// TIA Portal V17 export
// export: Created 2025-03-05T08:03:03.1395906Z, ExportSetting WithDefaults, DisplayName Totally Integrated Automation Portal, DisplayVersion V17 Update 8, DisplayName TIA Portal Openness, DisplayVersion V17 Update 8, DisplayName TIA Portal Version Control Interface, DisplayVersion V17, DisplayName SINAMICS Startdrive Advanced, DisplayVersion V17 SP2, DisplayName SINAMICS Startdrive G110M, G120, G120C, G120D, G120P, G115D, DisplayVersion V17 SP2, DisplayName SINAMICS Startdrive G130, G150, S120, S150, SINAMICS MV, S210, DisplayVersion V17 SP2, DisplayName STEP 7 Professional, DisplayVersion V17 Update 8, DisplayName SINUMERIK ONE STEP 7 Toolbox, DisplayVersion V17 Update 12, DisplayName SINUMERIK 840D sl STEP 7 Toolbox, DisplayVersion V17 Update 12, DisplayName STEP 7 Safety, DisplayVersion V17 Update 6, DisplayName WinCC Advanced, DisplayVersion V17 Update 8
FUNCTION_BLOCK "FB21013_POWDER_FEEDER_HOPPER"   // FB21013, LAD
TITLE = FB21013 POWDER FEEDER HOPPER
{ S7_Optimized_Access := 'FALSE' }
VERSION : 0.1
// stored: AutoNumber false, IsIECCheckEnabled false, SetENOAutomatically false, UDAEnableTagReadback false
   VAR_INPUT
      OPTIONS_0 : Byte := 2#0000_0000;
      iGENERAL_CONDITIONS : Bool;   // GENERAL CONDITIONS
      iPF_LINE_1_NOT_READY_FAULT : Bool;   // PF NOT READY FAULT LINE 1
      iPF_PROFINET_MODE_ACTIVE_FAULT_LINE_1 : Bool;   // PF PROFINET MODE ACTIVE FAULT LINE 1
      iPF_LINE_2_NOT_READY_FAULT : Bool;   // PF NOT READY FAULT LINE 2
      iMANUAL_START_REQ_LINE_1 : Bool;
      iMANUAL_START_REQ_LINE_2 : Bool;
      iMANUAL_STOP_REQ_LINE_1 : Bool;
      iMANUAL_STOP_REQ_LINE_2 : Bool;
      iPF_INTERLOCK_INPUTS : "POWDER FEEDER INTERLOCK INPUT";
      iFEEDER_PROFINET_MODE_ACTIVE : Bool;
      iCONTROL_ON_DELAYED : Bool;   // LOCAL MACHINE ON
      iAUTO_START_REQUEST : Bool;
      iAUTO_STOP_REQUEST : Bool;
      iHMI_GAS_SETPOINT_L1 : Real;
      iHMI_GAS_SETPOINT_L2 : Real;
      iHMI_DISK_SETPOINT_L1 : Real;
      iHMI_DISK_SETPOINT_L2 : Real;
      iCNC_GAS_SETPOINT_L1 : Real;
      iCNC_GAS_SETPOINT_L2 : Real;
      iCNC_DISK_SETPOINT_L1 : Real;
      iCNC_DISK_SETPOINT_L2 : Real;
      iFEEDER_PLC_AUX_VALUES : "POWDER FEEDER PLC AUXILIAR";
   END_VAR
   VAR_OUTPUT
      oSTATION_IS_ALARMS : Bool;   // STATION IS ALARMS
      oSTATION_WARNINGS : Bool;   // STATION WARNINGS
      o_fShutdownToPF_Line1 { ExternalAccessible := 'False'; ExternalVisible := 'False'; ExternalWritable := 'False'} : Bool;
      o_fShutdownToPF_Line2 { ExternalAccessible := 'False'; ExternalVisible := 'False'; ExternalWritable := 'False'} : Bool;
      o_fFeedingAllOnCmd_Line1 { ExternalAccessible := 'False'; ExternalVisible := 'False'; ExternalWritable := 'False'} : Bool;
      o_fFeedingAllOnCmd_Line2 { ExternalAccessible := 'False'; ExternalVisible := 'False'; ExternalWritable := 'False'} : Bool;
      o_fCarriergasOnCmd_Line1 { ExternalAccessible := 'False'; ExternalVisible := 'False'; ExternalWritable := 'False'} : Bool;
      o_fCarriergasOnCmd_Line2 { ExternalAccessible := 'False'; ExternalVisible := 'False'; ExternalWritable := 'False'} : Bool;
      o_fFeedingAllOffCmd_Line1 { ExternalAccessible := 'False'; ExternalVisible := 'False'; ExternalWritable := 'False'} : Bool;
      o_fFeedingAllOffCmd_Line2 { ExternalAccessible := 'False'; ExternalVisible := 'False'; ExternalWritable := 'False'} : Bool;
      o_fCarriergasOffCmd_Line1 { ExternalAccessible := 'False'; ExternalVisible := 'False'; ExternalWritable := 'False'} : Bool;
      o_fCarriergasOffCmd_Line2 { ExternalAccessible := 'False'; ExternalVisible := 'False'; ExternalWritable := 'False'} : Bool;
      oALARM_POWDER_LINE_1_CLOGGED : Bool;   // ALARM POWDER LINE 1 CLOGGED
      oALARM_GAS_FLOW_BELOW_LOW_LIMIT_LN_1 : Bool;   // ALARM GAS FLOW BELOW LOW LIMIT LINE 1
      oALARM_DISK_SPEED_BELOW_LOW_LIMIT_LN_1 : Bool;   // ALARM DISK SPEED BELOW LOW LIMIT LINE 1
      oALARM_STIRRER_SPEED_BELOW_LOW_LIMIT_LN_1 : Bool;   // ALARM STIRRER SPEED BELOW LOW LIMIT LINE 1
      oALARM_GAS_FLOW_ABOVE_HIGH_LIMIT_LN_1 : Bool;   // ALARM GAS FLOW ABOVE HIGH LIMIT LINE 1
      oALARM_DISK_SPEED_ABOVE_HIGH_LIMIT_LN_1 : Bool;   // ALARM DISK SPEED ABOVE HIGH LIMIT LINE 1
      oALARM_STIRRER_SPEED_ABOVE_HIGH_LIMIT_LN_1 : Bool;   // ALARM STIRRER SPEED ABOVE HIGH LIMIT LINE 1
      oALARM_CARRIER_GAS_INLET_PRESSURE_TOO_LOW_LN_1 : Bool;   // ALARM CARRIER GAS INLET PRESSURE TOO LOW LINE 1
      oALARM_DISK_MOTOR_PLUGGED_IN_AND_READY_LN_1 : Bool;   // ALARM DISK MOTOR PLUGGED IN AND READY LINE 1
      oALARM_STIRRER_PLUGGED_IN_AND_READY_LN_1 : Bool;   // ALARM STIRRER PLUGGED IN AND READY LINE 1
      oALARM_COMMUNICATION_RUNNING_LN_1 : Bool;   // ALARM COMMUNICATION RUNNING LINE 1
      oALARM_FEEDER_NOT_READY_LN_1 : Bool;   // ALARM FEEDER NOT READY LINE 1
      oWARNING_GAS_FLOW_UNDER_LIMIT_LN_1 : Bool;   // WARNING GAS FLOW UNDER LIMIT LINE 1
      oWARNING_DISK_SPEED_UNDER_LIMIT_LN_1 : Bool;   // WARNING DISK SPEED UNDER LIMIT LINE 1
      oWARNING_STIRRER_SPEED_UNDER_LIMIT_LN_1 : Bool;   // WARNING STIRRER SPEED UNDER LIMIT LINE 1
      oWARNING_GAS_FLOW_OVER_LIMIT_LN_1 : Bool;   // WARNING GAS FLOW OVER LIMIT LINE 1
      oWARNING_DISK_SPEED_OVER_LIMIT_LN_1 : Bool;   // WARNING DISK SPEED OVER LIMIT LINE 1
      oWARNING_STIRRER_SPEED_OVER_LIMIT_LN_1 : Bool;   // WARNING STIRRER SPEED OVER LIMIT LINE 1
      oALARM_POWDER_LINE_2_CLOGGED : Bool;   // ALARM POWDER LINE 2 CLOGGED
      oALARM_GAS_FLOW_BELOW_LOW_LIMIT_LN_2 : Bool;   // ALARM GAS FLOW BELOW LOW LIMIT LINE 2
      oALARM_DISK_SPEED_BELOW_LOW_LIMIT_LN_2 : Bool;   // ALARM DISK SPEED BELOW LOW LIMIT LINE 2
      oALARM_STIRRER_SPEED_BELOW_LOW_LIMIT_LN_2 : Bool;   // ALARM STIRRER SPEED BELOW LOW LIMIT LINE 2
      oALARM_GAS_FLOW_ABOVE_HIGH_LIMIT_LN_2 : Bool;   // ALARM GAS FLOW ABOVE HIGH LIMIT LINE 2
      oALARM_DISK_SPEED_ABOVE_HIGH_LIMIT_LN_2 : Bool;   // ALARM DISK SPEED ABOVE HIGH LIMIT LINE 2
      oALARM_STIRRER_SPEED_ABOVE_HIGH_LIMIT_LN_2 : Bool;   // ALARM STIRRER SPEED ABOVE HIGH LIMIT LINE 2
      oALARM_CARRIER_GAS_INLET_PRESSURE_TOO_LOW_LN_2 : Bool;   // ALARM CARRIER GAS INLET PRESSURE TOO LOW LINE 2
      oALARM_DISK_MOTOR_PLUGGED_IN_AND_READY_LN_2 : Bool;   // ALARM DISK MOTOR PLUGGED IN AND READY LINE 2
      oALARM_STIRRER_PLUGGED_IN_AND_READY_LN_2 : Bool;   // ALARM STIRRER PLUGGED IN AND READY LINE 2
      oALARM_COMMUNICATION_RUNNING_LN_2 : Bool;   // ALARM COMMUNICATION RUNNING LINE 2
      oALARM_FEEDER_NOT_READY_LN_2 : Bool;   // ALARM FEEDER NOT READY LINE 2
      oWARNING_GAS_FLOW_UNDER_LIMIT_LN_2 : Bool;   // WARNING GAS FLOW UNDER LIMIT LINE 2
      oWARNING_DISK_SPEED_UNDER_LIMIT_LN_2 : Bool;   // WARNING DISK SPEED UNDER LIMIT LINE 2
      oWARNING_STIRRER_SPEED_UNDER_LIMIT_LN_2 : Bool;   // WARNING STIRRER SPEED UNDER LIMIT LINE 2
      oWARNING_GAS_FLOW_OVER_LIMIT_LN_2 : Bool;   // WARNING GAS FLOW OVER LIMIT LINE 2
      oWARNING_DISK_SPEED_OVER_LIMIT_LN_2 : Bool;   // WARNING DISK SPEED OVER LIMIT LINE 2
      oWARNING_STIRRER_SPEED_OVER_LIMIT_LN_2 : Bool;   // WARNING STIRRER SPEED OVER LIMIT LINE 2
   END_VAR
   VAR DB_SPECIFIC
      DATA : "POWDER FEEDER HOPPER";
      INPUT_SETTINGS : Struct
         UNIT_NUMBER : Int;
         FEEDER_NUMBER : Int;
      END_STRUCT;
      Fault_timer { S7_SetPoint := 'True'} : TON_TIME;
      START_DONE_LINE_1 { S7_SetPoint := 'True'} : Bool;   // START DONE LINE 1
      START_DONE_LINE_2 { S7_SetPoint := 'True'} : Bool;   // START DONE LINE 2
      STOP_SEQUENCE_ON { S7_SetPoint := 'True'} : Bool;   // HOPPER STOP SEQUENCE IS ON
      STOP_PULSE_LINE_1 : Bool;
      STOP_PULSE_LINE_2 : Bool;
      HOPPER_STATUS_LINE_1 : Byte;   // HOPPER LINE 1 STATUS
      HOPPER_STATUS_LINE_2 : Byte;   // HOPPER LINE 2 STATUS
   END_VAR
   VAR
      SWITCH_ON_SEQUENCE_LINE_1 : "FB21250_POWDER_ON_OFF_SEQUENCE";
      SWITCH_ON_SEQUENCE_LINE_2 : "FB21250_POWDER_ON_OFF_SEQUENCE";
      SWITCH_OFF_SEQUENCE_LINE_1 : "FB21250_POWDER_ON_OFF_SEQUENCE";
      SWITCH_OFF_SEQUENCE_LINE_2 : "FB21250_POWDER_ON_OFF_SEQUENCE";
   END_VAR
   VAR DB_SPECIFIC
      SWITCH_OFF_DELAY_LINE_1 { S7_SetPoint := 'True'} : TOF_TIME;
      SWITCH_OFF_DELAY_LINE_2 { S7_SetPoint := 'True'} : TOF_TIME;
   END_VAR
   VAR_TEMP
      DB_NUMBER : DInt;
      INPUTS_MASK : Byte;
      O_BYTE_0 : Struct
         LINE_1_ENABLED : Bool;
         LINE_2_ENABLED : Bool;
         SPARE : Bool;
         SPARE_1 : Bool;
         SPARE_2 : Bool;
         SPARE_3 : Bool;
         SPARE_4 : Bool;
         SPARE_5 : Bool;
      END_STRUCT;
   END_VAR
   // Fault_timer.PT := T#1s;
   // SWITCH_OFF_DELAY_LINE_1.PT := T#4s;
   // SWITCH_OFF_DELAY_LINE_2.PT := T#4s;
   VAR_TEMP   // added for the SCL form of the ladder/FBD networks
      _w1 : Bool;
      _w2 : Bool;
   END_VAR
BEGIN

NETWORK
TITLE = READ INSTANCE DB NUMBER
      L     DINO;
      +     10#800000;
      T     #DB_NUMBER;

REGION Network 2: OPTIONS
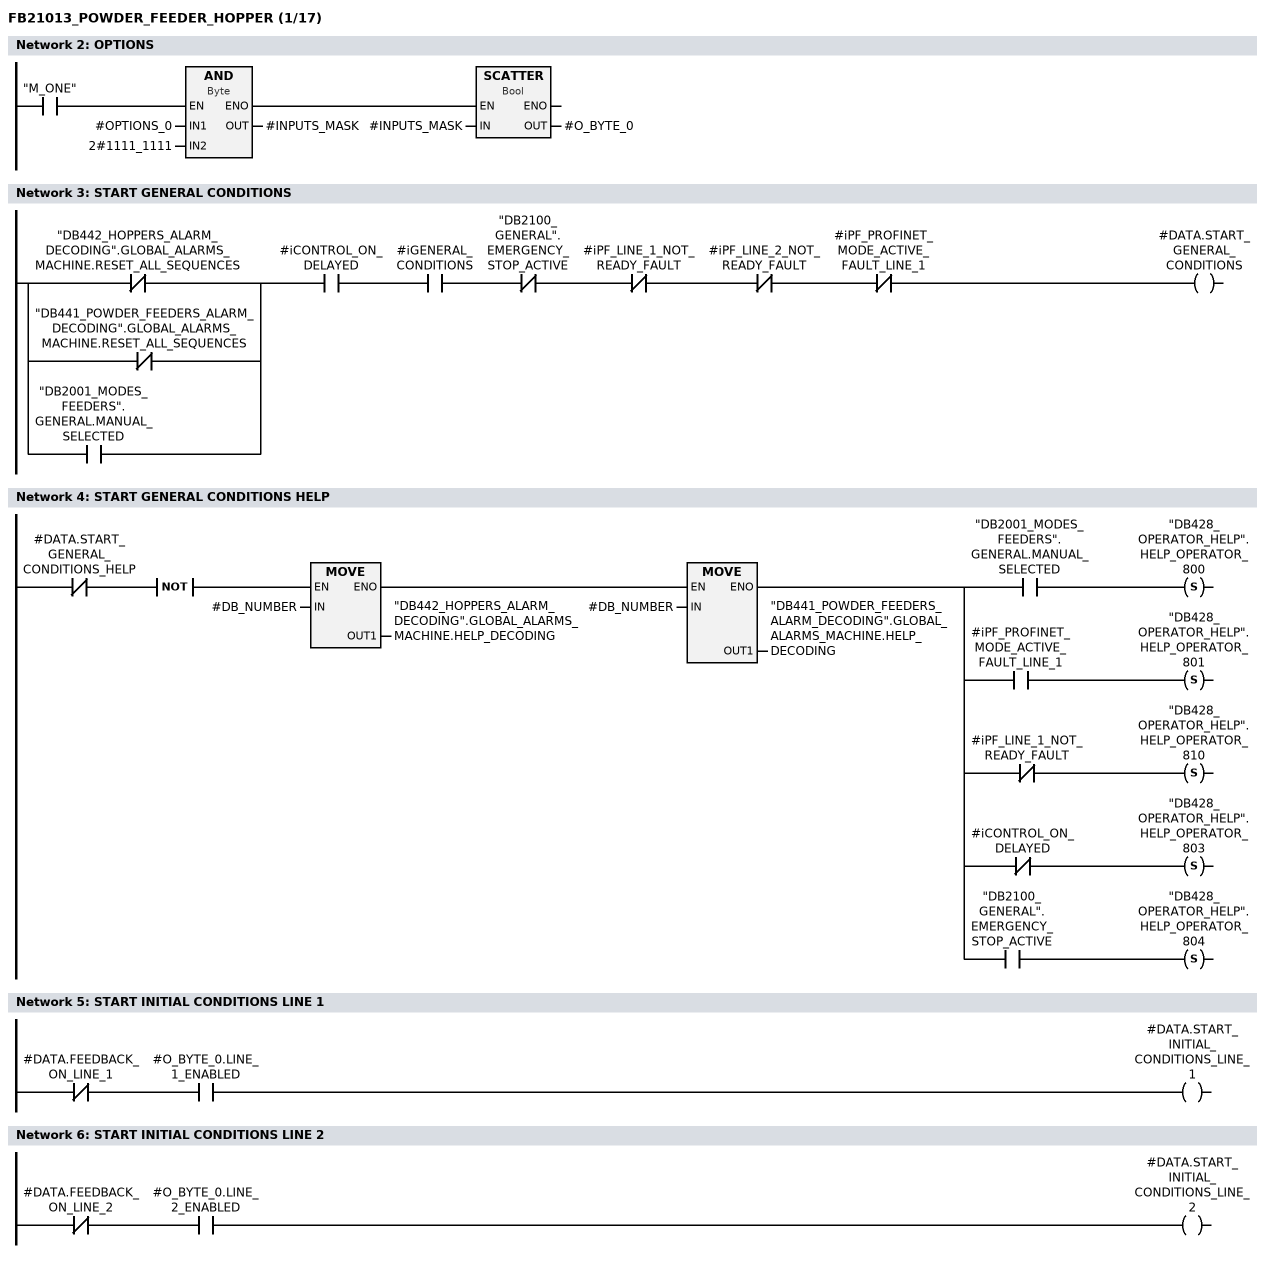
   RUNG wire#powerrail
      Contact( "M_ONE" )
      { S7_Templates := "SrcType := Byte" } And(in1 := #OPTIONS_0, in2 := 2#1111_1111, out => #INPUTS_MASK)
      { S7_Templates := "[dest_type := Bool, src_type := Byte]" } SCATTER(IN := #INPUTS_MASK, OUT => #O_BYTE_0)
   END_RUNG
   // the same network as SCL:
   IF "M_ONE" THEN
       #INPUTS_MASK := #OPTIONS_0 AND 2#1111_1111;
       SCATTER(IN := #INPUTS_MASK, OUT => #O_BYTE_0);
   END_IF;
END_REGION

REGION Network 3: START GENERAL CONDITIONS
   RUNG wire#powerrail
      I_Contact( "DB442_HOPPERS_ALARM_DECODING".GLOBAL_ALARMS_MACHINE.RESET_ALL_SEQUENCES )
      wire#w1
      Contact( #iCONTROL_ON_DELAYED )
      Contact( #iGENERAL_CONDITIONS )
      I_Contact( "DB2100_GENERAL".EMERGENCY_STOP_ACTIVE )
      I_Contact( #iPF_LINE_1_NOT_READY_FAULT )
      I_Contact( #iPF_LINE_2_NOT_READY_FAULT )
      I_Contact( #iPF_PROFINET_MODE_ACTIVE_FAULT_LINE_1 )
      Coil( #DATA.START_GENERAL_CONDITIONS )
   END_RUNG
   RUNG wire#powerrail
      I_Contact( "DB441_POWDER_FEEDERS_ALARM_DECODING".GLOBAL_ALARMS_MACHINE.RESET_ALL_SEQUENCES )
   END_RUNG wire#w1
   RUNG wire#powerrail
      Contact( "DB2001_MODES_FEEDERS".GENERAL.MANUAL_SELECTED )
   END_RUNG wire#w1
   // the same network as SCL:
   #DATA.START_GENERAL_CONDITIONS := (NOT "DB442_HOPPERS_ALARM_DECODING".GLOBAL_ALARMS_MACHINE.RESET_ALL_SEQUENCES OR NOT "DB441_POWDER_FEEDERS_ALARM_DECODING".GLOBAL_ALARMS_MACHINE.RESET_ALL_SEQUENCES OR "DB2001_MODES_FEEDERS".GENERAL.MANUAL_SELECTED) AND #iCONTROL_ON_DELAYED AND #iGENERAL_CONDITIONS AND NOT "DB2100_GENERAL".EMERGENCY_STOP_ACTIVE AND NOT #iPF_LINE_1_NOT_READY_FAULT AND NOT #iPF_LINE_2_NOT_READY_FAULT AND NOT #iPF_PROFINET_MODE_ACTIVE_FAULT_LINE_1;
END_REGION

REGION Network 4: START GENERAL CONDITIONS HELP
   RUNG wire#powerrail
      I_Contact( #DATA.START_GENERAL_CONDITIONS_HELP )
      Not()
      Move(in := #DB_NUMBER, out1 => "DB442_HOPPERS_ALARM_DECODING".GLOBAL_ALARMS_MACHINE.HELP_DECODING)
      Move(in := #DB_NUMBER, out1 => "DB441_POWDER_FEEDERS_ALARM_DECODING".GLOBAL_ALARMS_MACHINE.HELP_DECODING)
      wire#w1
      Contact( "DB2001_MODES_FEEDERS".GENERAL.MANUAL_SELECTED )
      S_Coil( "DB428_OPERATOR_HELP".HELP_OPERATOR_800 )
   END_RUNG
   RUNG wire#w1
      Contact( #iPF_PROFINET_MODE_ACTIVE_FAULT_LINE_1 )
      S_Coil( "DB428_OPERATOR_HELP".HELP_OPERATOR_801 )
   END_RUNG
   RUNG wire#w1
      I_Contact( #iPF_LINE_1_NOT_READY_FAULT )
      S_Coil( "DB428_OPERATOR_HELP".HELP_OPERATOR_810 )
   END_RUNG
   RUNG wire#w1
      I_Contact( #iCONTROL_ON_DELAYED )
      S_Coil( "DB428_OPERATOR_HELP".HELP_OPERATOR_803 )
   END_RUNG
   RUNG wire#w1
      Contact( "DB2100_GENERAL".EMERGENCY_STOP_ACTIVE )
      S_Coil( "DB428_OPERATOR_HELP".HELP_OPERATOR_804 )
   END_RUNG
   // the same network as SCL:
   #_w1 := NOT (NOT #DATA.START_GENERAL_CONDITIONS_HELP);
   IF #_w1 THEN
       "DB442_HOPPERS_ALARM_DECODING".GLOBAL_ALARMS_MACHINE.HELP_DECODING := #DB_NUMBER;
       "DB441_POWDER_FEEDERS_ALARM_DECODING".GLOBAL_ALARMS_MACHINE.HELP_DECODING := #DB_NUMBER;
   END_IF;
   IF #_w1 AND "DB2001_MODES_FEEDERS".GENERAL.MANUAL_SELECTED THEN
       "DB428_OPERATOR_HELP".HELP_OPERATOR_800 := TRUE;
   END_IF;
   IF #_w1 AND #iPF_PROFINET_MODE_ACTIVE_FAULT_LINE_1 THEN
       "DB428_OPERATOR_HELP".HELP_OPERATOR_801 := TRUE;
   END_IF;
   IF #_w1 AND NOT #iPF_LINE_1_NOT_READY_FAULT THEN "DB428_OPERATOR_HELP".HELP_OPERATOR_810 := TRUE; END_IF;
   IF #_w1 AND NOT #iCONTROL_ON_DELAYED THEN "DB428_OPERATOR_HELP".HELP_OPERATOR_803 := TRUE; END_IF;
   IF #_w1 AND "DB2100_GENERAL".EMERGENCY_STOP_ACTIVE THEN
       "DB428_OPERATOR_HELP".HELP_OPERATOR_804 := TRUE;
   END_IF;
END_REGION

REGION Network 5: START INITIAL CONDITIONS LINE 1
   RUNG wire#powerrail
      I_Contact( #DATA.FEEDBACK_ON_LINE_1 )
      Contact( #O_BYTE_0.LINE_1_ENABLED )
      Coil( #DATA.START_INITIAL_CONDITIONS_LINE_1 )
   END_RUNG
   // the same network as SCL:
   #DATA.START_INITIAL_CONDITIONS_LINE_1 := NOT #DATA.FEEDBACK_ON_LINE_1 AND #O_BYTE_0.LINE_1_ENABLED;
END_REGION

REGION Network 6: START INITIAL CONDITIONS LINE 2
   RUNG wire#powerrail
      I_Contact( #DATA.FEEDBACK_ON_LINE_2 )
      Contact( #O_BYTE_0.LINE_2_ENABLED )
      Coil( #DATA.START_INITIAL_CONDITIONS_LINE_2 )
   END_RUNG
   // the same network as SCL:
   #DATA.START_INITIAL_CONDITIONS_LINE_2 := NOT #DATA.FEEDBACK_ON_LINE_2 AND #O_BYTE_0.LINE_2_ENABLED;
END_REGION

REGION Network 7: START INITIAL CONDITIONS HELP
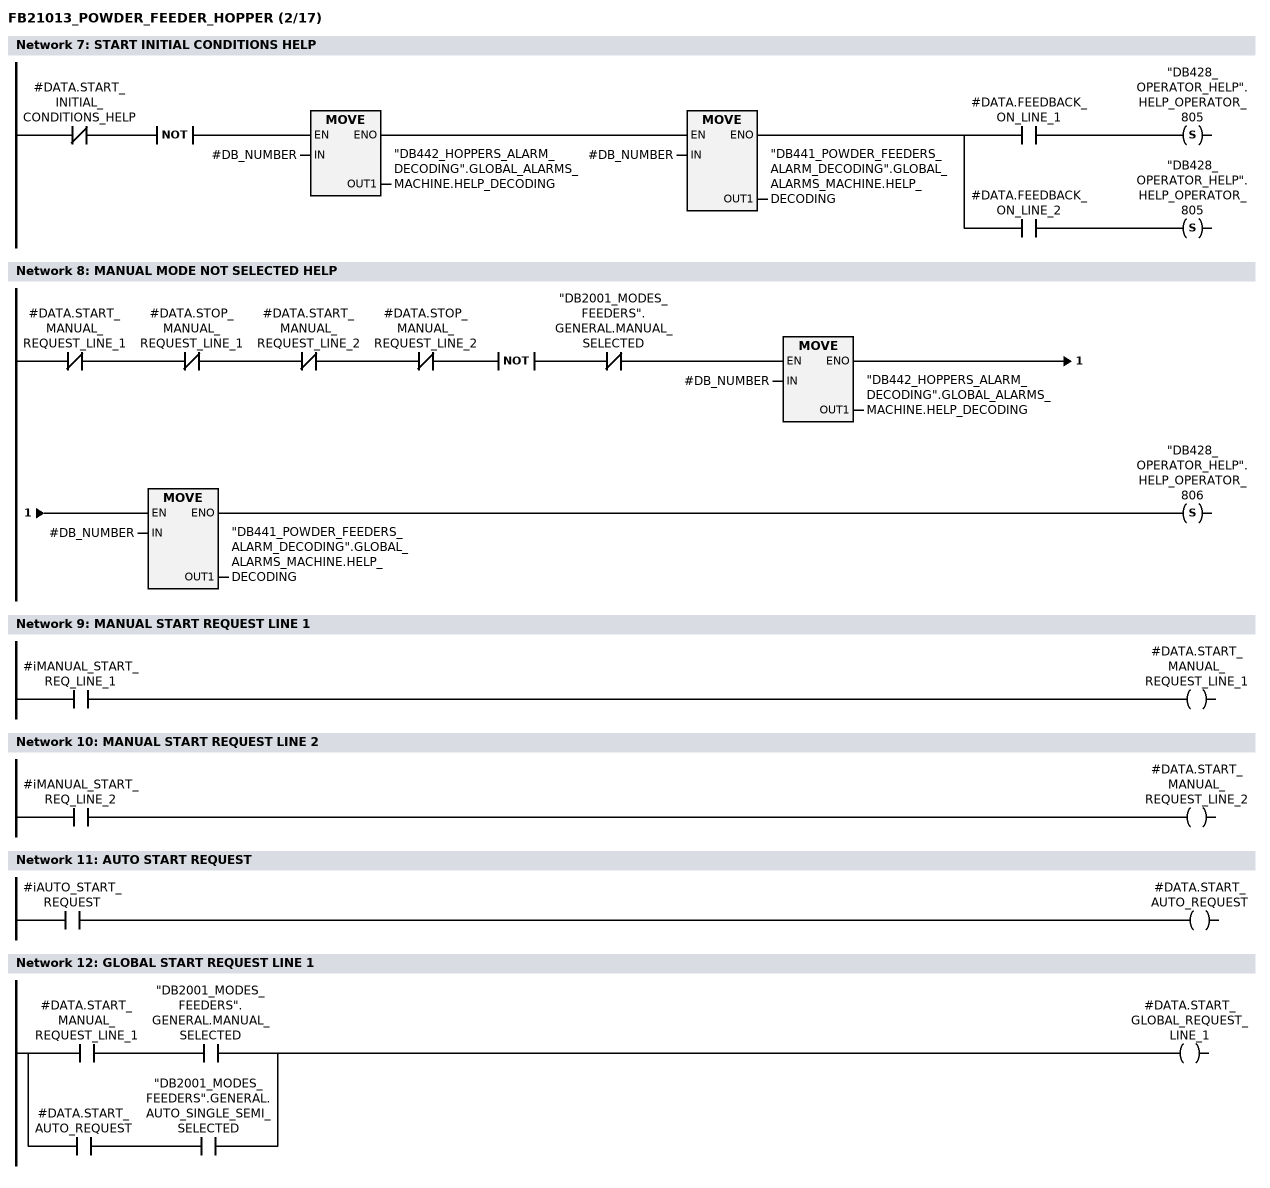
   RUNG wire#powerrail
      I_Contact( #DATA.START_INITIAL_CONDITIONS_HELP )
      Not()
      Move(in := #DB_NUMBER, out1 => "DB442_HOPPERS_ALARM_DECODING".GLOBAL_ALARMS_MACHINE.HELP_DECODING)
      Move(in := #DB_NUMBER, out1 => "DB441_POWDER_FEEDERS_ALARM_DECODING".GLOBAL_ALARMS_MACHINE.HELP_DECODING)
      wire#w1
      Contact( #DATA.FEEDBACK_ON_LINE_1 )
      S_Coil( "DB428_OPERATOR_HELP".HELP_OPERATOR_805 )
   END_RUNG
   RUNG wire#w1
      Contact( #DATA.FEEDBACK_ON_LINE_2 )
      S_Coil( "DB428_OPERATOR_HELP".HELP_OPERATOR_805 )
   END_RUNG
   // the same network as SCL:
   #_w1 := NOT (NOT #DATA.START_INITIAL_CONDITIONS_HELP);
   IF #_w1 THEN
       "DB442_HOPPERS_ALARM_DECODING".GLOBAL_ALARMS_MACHINE.HELP_DECODING := #DB_NUMBER;
       "DB441_POWDER_FEEDERS_ALARM_DECODING".GLOBAL_ALARMS_MACHINE.HELP_DECODING := #DB_NUMBER;
   END_IF;
   IF #_w1 AND #DATA.FEEDBACK_ON_LINE_1 THEN "DB428_OPERATOR_HELP".HELP_OPERATOR_805 := TRUE; END_IF;
   IF #_w1 AND #DATA.FEEDBACK_ON_LINE_2 THEN "DB428_OPERATOR_HELP".HELP_OPERATOR_805 := TRUE; END_IF;
END_REGION

REGION Network 8: MANUAL MODE NOT SELECTED HELP
   RUNG wire#powerrail
      I_Contact( #DATA.START_MANUAL_REQUEST_LINE_1 )
      I_Contact( #DATA.STOP_MANUAL_REQUEST_LINE_1 )
      I_Contact( #DATA.START_MANUAL_REQUEST_LINE_2 )
      I_Contact( #DATA.STOP_MANUAL_REQUEST_LINE_2 )
      Not()
      I_Contact( "DB2001_MODES_FEEDERS".GENERAL.MANUAL_SELECTED )
      Move(in := #DB_NUMBER, out1 => "DB442_HOPPERS_ALARM_DECODING".GLOBAL_ALARMS_MACHINE.HELP_DECODING)
      Move(in := #DB_NUMBER, out1 => "DB441_POWDER_FEEDERS_ALARM_DECODING".GLOBAL_ALARMS_MACHINE.HELP_DECODING)
      S_Coil( "DB428_OPERATOR_HELP".HELP_OPERATOR_806 )
   END_RUNG
   // the same network as SCL:
   IF NOT (NOT #DATA.START_MANUAL_REQUEST_LINE_1 AND NOT #DATA.STOP_MANUAL_REQUEST_LINE_1 AND NOT #DATA.START_MANUAL_REQUEST_LINE_2 AND NOT #DATA.STOP_MANUAL_REQUEST_LINE_2) AND NOT "DB2001_MODES_FEEDERS".GENERAL.MANUAL_SELECTED THEN
       "DB442_HOPPERS_ALARM_DECODING".GLOBAL_ALARMS_MACHINE.HELP_DECODING := #DB_NUMBER;
       "DB441_POWDER_FEEDERS_ALARM_DECODING".GLOBAL_ALARMS_MACHINE.HELP_DECODING := #DB_NUMBER;
       "DB428_OPERATOR_HELP".HELP_OPERATOR_806 := TRUE;
   END_IF;
END_REGION

REGION Network 9: MANUAL START REQUEST LINE 1
   RUNG wire#powerrail
      Contact( #iMANUAL_START_REQ_LINE_1 )
      Coil( #DATA.START_MANUAL_REQUEST_LINE_1 )
   END_RUNG
   // the same network as SCL:
   #DATA.START_MANUAL_REQUEST_LINE_1 := #iMANUAL_START_REQ_LINE_1;
END_REGION

REGION Network 10: MANUAL START REQUEST LINE 2
   RUNG wire#powerrail
      Contact( #iMANUAL_START_REQ_LINE_2 )
      Coil( #DATA.START_MANUAL_REQUEST_LINE_2 )
   END_RUNG
   // the same network as SCL:
   #DATA.START_MANUAL_REQUEST_LINE_2 := #iMANUAL_START_REQ_LINE_2;
END_REGION

REGION Network 11: AUTO START REQUEST
   RUNG wire#powerrail
      Contact( #iAUTO_START_REQUEST )
      Coil( #DATA.START_AUTO_REQUEST )
   END_RUNG
   // the same network as SCL:
   #DATA.START_AUTO_REQUEST := #iAUTO_START_REQUEST;
END_REGION

REGION Network 12: GLOBAL START REQUEST LINE 1
   RUNG wire#powerrail
      Contact( #DATA.START_MANUAL_REQUEST_LINE_1 )
      Contact( "DB2001_MODES_FEEDERS".GENERAL.MANUAL_SELECTED )
      wire#w1
      Coil( #DATA.START_GLOBAL_REQUEST_LINE_1 )
   END_RUNG
   RUNG wire#powerrail
      Contact( #DATA.START_AUTO_REQUEST )
      Contact( "DB2001_MODES_FEEDERS".GENERAL.AUTO_SINGLE_SEMI_SELECTED )
   END_RUNG wire#w1
   // the same network as SCL:
   #DATA.START_GLOBAL_REQUEST_LINE_1 := (#DATA.START_MANUAL_REQUEST_LINE_1 AND "DB2001_MODES_FEEDERS".GENERAL.MANUAL_SELECTED) OR (#DATA.START_AUTO_REQUEST AND "DB2001_MODES_FEEDERS".GENERAL.AUTO_SINGLE_SEMI_SELECTED);
END_REGION

REGION Network 13: GLOBAL START REQUEST LINE 2
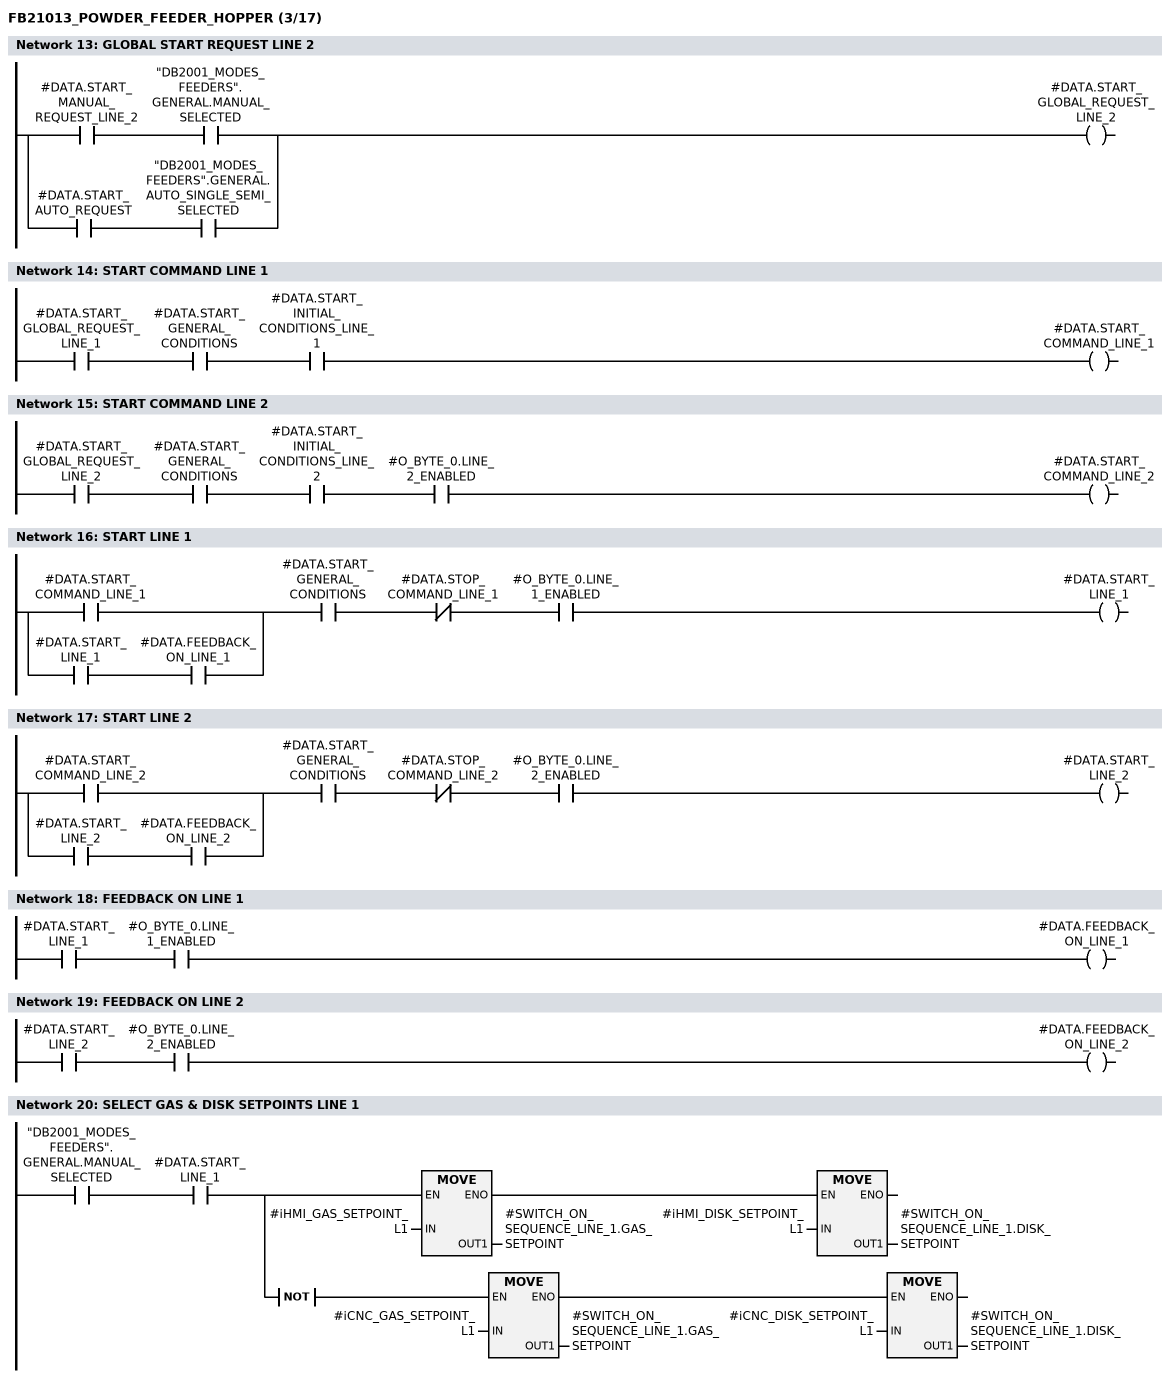
   RUNG wire#powerrail
      Contact( #DATA.START_MANUAL_REQUEST_LINE_2 )
      Contact( "DB2001_MODES_FEEDERS".GENERAL.MANUAL_SELECTED )
      wire#w1
      Coil( #DATA.START_GLOBAL_REQUEST_LINE_2 )
   END_RUNG
   RUNG wire#powerrail
      Contact( #DATA.START_AUTO_REQUEST )
      Contact( "DB2001_MODES_FEEDERS".GENERAL.AUTO_SINGLE_SEMI_SELECTED )
   END_RUNG wire#w1
   // the same network as SCL:
   #DATA.START_GLOBAL_REQUEST_LINE_2 := (#DATA.START_MANUAL_REQUEST_LINE_2 AND "DB2001_MODES_FEEDERS".GENERAL.MANUAL_SELECTED) OR (#DATA.START_AUTO_REQUEST AND "DB2001_MODES_FEEDERS".GENERAL.AUTO_SINGLE_SEMI_SELECTED);
END_REGION

REGION Network 14: START COMMAND LINE 1
   RUNG wire#powerrail
      Contact( #DATA.START_GLOBAL_REQUEST_LINE_1 )
      Contact( #DATA.START_GENERAL_CONDITIONS )
      Contact( #DATA.START_INITIAL_CONDITIONS_LINE_1 )
      Coil( #DATA.START_COMMAND_LINE_1 )
   END_RUNG
   // the same network as SCL:
   #DATA.START_COMMAND_LINE_1 := #DATA.START_GLOBAL_REQUEST_LINE_1 AND #DATA.START_GENERAL_CONDITIONS AND #DATA.START_INITIAL_CONDITIONS_LINE_1;
END_REGION

REGION Network 15: START COMMAND LINE 2
   RUNG wire#powerrail
      Contact( #DATA.START_GLOBAL_REQUEST_LINE_2 )
      Contact( #DATA.START_GENERAL_CONDITIONS )
      Contact( #DATA.START_INITIAL_CONDITIONS_LINE_2 )
      Contact( #O_BYTE_0.LINE_2_ENABLED )
      Coil( #DATA.START_COMMAND_LINE_2 )
   END_RUNG
   // the same network as SCL:
   #DATA.START_COMMAND_LINE_2 := #DATA.START_GLOBAL_REQUEST_LINE_2 AND #DATA.START_GENERAL_CONDITIONS AND #DATA.START_INITIAL_CONDITIONS_LINE_2 AND #O_BYTE_0.LINE_2_ENABLED;
END_REGION

REGION Network 16: START LINE 1
   RUNG wire#powerrail
      Contact( #DATA.START_COMMAND_LINE_1 )
      wire#w1
      Contact( #DATA.START_GENERAL_CONDITIONS )
      I_Contact( #DATA.STOP_COMMAND_LINE_1 )
      Contact( #O_BYTE_0.LINE_1_ENABLED )
      Coil( #DATA.START_LINE_1 )
   END_RUNG
   RUNG wire#powerrail
      Contact( #DATA.START_LINE_1 )
      Contact( #DATA.FEEDBACK_ON_LINE_1 )
   END_RUNG wire#w1
   // the same network as SCL:
   #DATA.START_LINE_1 := (#DATA.START_COMMAND_LINE_1 OR (#DATA.START_LINE_1 AND #DATA.FEEDBACK_ON_LINE_1)) AND #DATA.START_GENERAL_CONDITIONS AND NOT #DATA.STOP_COMMAND_LINE_1 AND #O_BYTE_0.LINE_1_ENABLED;
END_REGION

REGION Network 17: START LINE 2
   RUNG wire#powerrail
      Contact( #DATA.START_COMMAND_LINE_2 )
      wire#w1
      Contact( #DATA.START_GENERAL_CONDITIONS )
      I_Contact( #DATA.STOP_COMMAND_LINE_2 )
      Contact( #O_BYTE_0.LINE_2_ENABLED )
      Coil( #DATA.START_LINE_2 )
   END_RUNG
   RUNG wire#powerrail
      Contact( #DATA.START_LINE_2 )
      Contact( #DATA.FEEDBACK_ON_LINE_2 )
   END_RUNG wire#w1
   // the same network as SCL:
   #DATA.START_LINE_2 := (#DATA.START_COMMAND_LINE_2 OR (#DATA.START_LINE_2 AND #DATA.FEEDBACK_ON_LINE_2)) AND #DATA.START_GENERAL_CONDITIONS AND NOT #DATA.STOP_COMMAND_LINE_2 AND #O_BYTE_0.LINE_2_ENABLED;
END_REGION

REGION Network 18: FEEDBACK ON LINE 1
   RUNG wire#powerrail
      Contact( #DATA.START_LINE_1 )
      Contact( #O_BYTE_0.LINE_1_ENABLED )
      Coil( #DATA.FEEDBACK_ON_LINE_1 )
   END_RUNG
   // the same network as SCL:
   #DATA.FEEDBACK_ON_LINE_1 := #DATA.START_LINE_1 AND #O_BYTE_0.LINE_1_ENABLED;
END_REGION

REGION Network 19: FEEDBACK ON LINE 2
   RUNG wire#powerrail
      Contact( #DATA.START_LINE_2 )
      Contact( #O_BYTE_0.LINE_2_ENABLED )
      Coil( #DATA.FEEDBACK_ON_LINE_2 )
   END_RUNG
   // the same network as SCL:
   #DATA.FEEDBACK_ON_LINE_2 := #DATA.START_LINE_2 AND #O_BYTE_0.LINE_2_ENABLED;
END_REGION

REGION Network 20: SELECT GAS & DISK SETPOINTS LINE 1
   RUNG wire#powerrail
      Contact( "DB2001_MODES_FEEDERS".GENERAL.MANUAL_SELECTED )
      Contact( #DATA.START_LINE_1 )
      wire#w1
      Move(in := #iHMI_GAS_SETPOINT_L1, out1 => #SWITCH_ON_SEQUENCE_LINE_1.GAS_SETPOINT)
      Move(in := #iHMI_DISK_SETPOINT_L1, out1 => #SWITCH_ON_SEQUENCE_LINE_1.DISK_SETPOINT)
   END_RUNG
   RUNG wire#w1
      Not()
      Move(in := #iCNC_GAS_SETPOINT_L1, out1 => #SWITCH_ON_SEQUENCE_LINE_1.GAS_SETPOINT)
      Move(in := #iCNC_DISK_SETPOINT_L1, out1 => #SWITCH_ON_SEQUENCE_LINE_1.DISK_SETPOINT)
   END_RUNG
   // the same network as SCL:
   #_w1 := "DB2001_MODES_FEEDERS".GENERAL.MANUAL_SELECTED AND #DATA.START_LINE_1;
   IF #_w1 THEN
       #SWITCH_ON_SEQUENCE_LINE_1.GAS_SETPOINT := #iHMI_GAS_SETPOINT_L1;
       #SWITCH_ON_SEQUENCE_LINE_1.DISK_SETPOINT := #iHMI_DISK_SETPOINT_L1;
   END_IF;
   IF NOT #_w1 THEN
       #SWITCH_ON_SEQUENCE_LINE_1.GAS_SETPOINT := #iCNC_GAS_SETPOINT_L1;
       #SWITCH_ON_SEQUENCE_LINE_1.DISK_SETPOINT := #iCNC_DISK_SETPOINT_L1;
   END_IF;
END_REGION

REGION Network 21: SELECT GAS & DISK SETPOINTS LINE 2
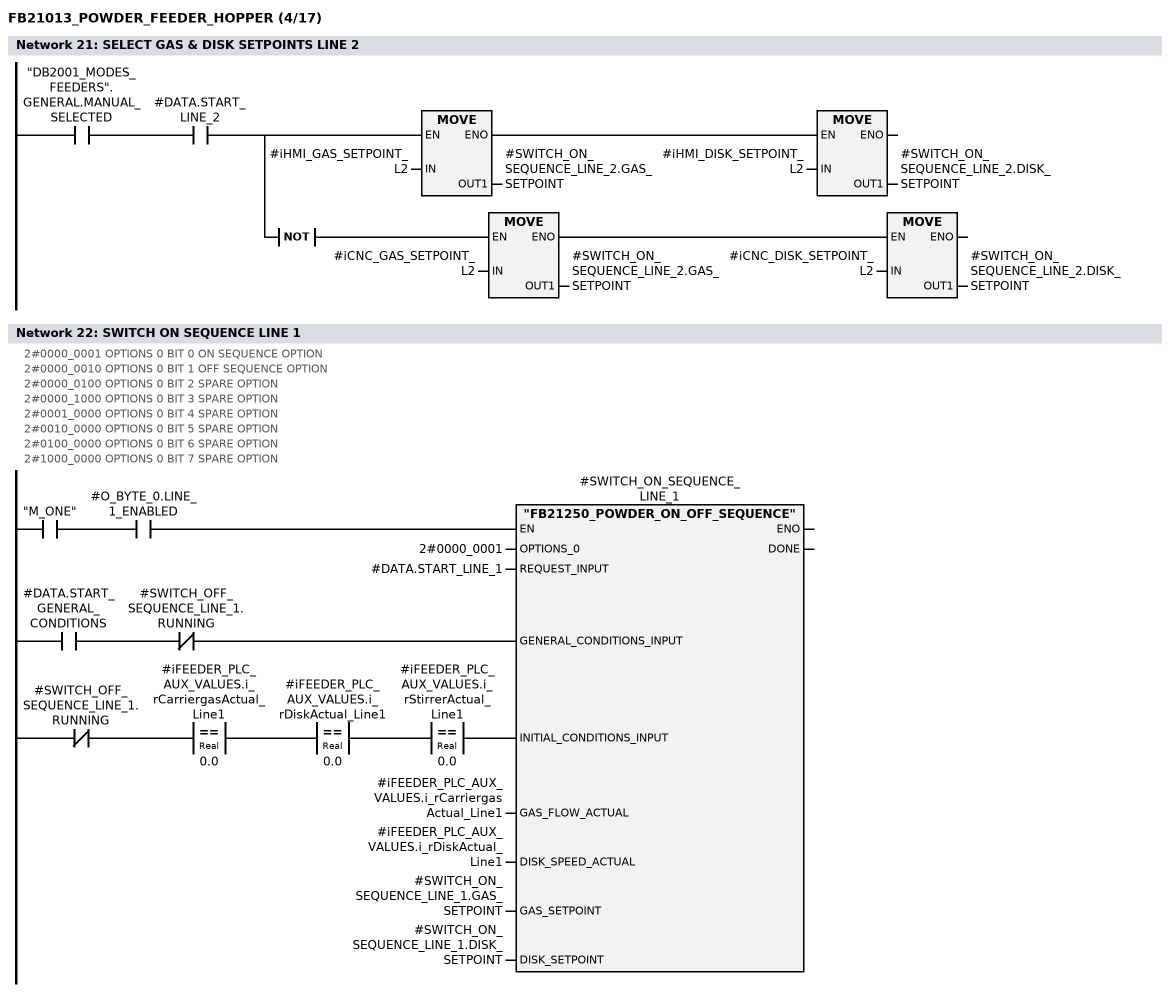
   RUNG wire#powerrail
      Contact( "DB2001_MODES_FEEDERS".GENERAL.MANUAL_SELECTED )
      Contact( #DATA.START_LINE_2 )
      wire#w1
      Move(in := #iHMI_GAS_SETPOINT_L2, out1 => #SWITCH_ON_SEQUENCE_LINE_2.GAS_SETPOINT)
      Move(in := #iHMI_DISK_SETPOINT_L2, out1 => #SWITCH_ON_SEQUENCE_LINE_2.DISK_SETPOINT)
   END_RUNG
   RUNG wire#w1
      Not()
      Move(in := #iCNC_GAS_SETPOINT_L2, out1 => #SWITCH_ON_SEQUENCE_LINE_2.GAS_SETPOINT)
      Move(in := #iCNC_DISK_SETPOINT_L2, out1 => #SWITCH_ON_SEQUENCE_LINE_2.DISK_SETPOINT)
   END_RUNG
   // the same network as SCL:
   #_w1 := "DB2001_MODES_FEEDERS".GENERAL.MANUAL_SELECTED AND #DATA.START_LINE_2;
   IF #_w1 THEN
       #SWITCH_ON_SEQUENCE_LINE_2.GAS_SETPOINT := #iHMI_GAS_SETPOINT_L2;
       #SWITCH_ON_SEQUENCE_LINE_2.DISK_SETPOINT := #iHMI_DISK_SETPOINT_L2;
   END_IF;
   IF NOT #_w1 THEN
       #SWITCH_ON_SEQUENCE_LINE_2.GAS_SETPOINT := #iCNC_GAS_SETPOINT_L2;
       #SWITCH_ON_SEQUENCE_LINE_2.DISK_SETPOINT := #iCNC_DISK_SETPOINT_L2;
   END_IF;
END_REGION

REGION Network 22: SWITCH ON SEQUENCE LINE 1
   // 2#0000_0001 OPTIONS 0 BIT 0 ON SEQUENCE OPTION
   // 2#0000_0010 OPTIONS 0 BIT 1 OFF SEQUENCE OPTION
   // 2#0000_0100 OPTIONS 0 BIT 2 SPARE OPTION
   // 2#0000_1000 OPTIONS 0 BIT 3 SPARE OPTION
   // 2#0001_0000 OPTIONS 0 BIT 4 SPARE OPTION
   // 2#0010_0000 OPTIONS 0 BIT 5 SPARE OPTION
   // 2#0100_0000 OPTIONS 0 BIT 6 SPARE OPTION
   // 2#1000_0000 OPTIONS 0 BIT 7 SPARE OPTION
   RUNG wire#powerrail
      Contact( "M_ONE" )
      Contact( #O_BYTE_0.LINE_1_ENABLED )
      #SWITCH_ON_SEQUENCE_LINE_1(GENERAL_CONDITIONS_INPUT := wire#w1, INITIAL_CONDITIONS_INPUT := wire#w2, OPTIONS_0 := 2#0000_0001, REQUEST_INPUT := #DATA.START_LINE_1, GAS_FLOW_ACTUAL := #iFEEDER_PLC_AUX_VALUES.i_rCarriergasActual_Line1, DISK_SPEED_ACTUAL := #iFEEDER_PLC_AUX_VALUES.i_rDiskActual_Line1, GAS_SETPOINT := #SWITCH_ON_SEQUENCE_LINE_1.GAS_SETPOINT, DISK_SETPOINT := #SWITCH_ON_SEQUENCE_LINE_1.DISK_SETPOINT, DONE =>)
   END_RUNG
   RUNG wire#powerrail
      Contact( #DATA.START_GENERAL_CONDITIONS )
      I_Contact( #SWITCH_OFF_SEQUENCE_LINE_1.RUNNING )
   END_RUNG wire#w1
   RUNG wire#powerrail
      I_Contact( #SWITCH_OFF_SEQUENCE_LINE_1.RUNNING )
      { S7_Templates := "SrcType := Real" } EQ_Contact(in1 := #iFEEDER_PLC_AUX_VALUES.i_rCarriergasActual_Line1, in2 := 0.0)
      { S7_Templates := "SrcType := Real" } EQ_Contact(in1 := #iFEEDER_PLC_AUX_VALUES.i_rDiskActual_Line1, in2 := 0.0)
      { S7_Templates := "SrcType := Real" } EQ_Contact(in1 := #iFEEDER_PLC_AUX_VALUES.i_rStirrerActual_Line1, in2 := 0.0)
   END_RUNG wire#w2
   // the same network as SCL:
   IF "M_ONE" AND #O_BYTE_0.LINE_1_ENABLED THEN
       #SWITCH_ON_SEQUENCE_LINE_1(OPTIONS_0 := 2#0000_0001,   // "FB21250_POWDER_ON_OFF_SEQUENCE"
                               REQUEST_INPUT := #DATA.START_LINE_1,
                               GENERAL_CONDITIONS_INPUT := #DATA.START_GENERAL_CONDITIONS AND NOT #SWITCH_OFF_SEQUENCE_LINE_1.RUNNING,
                               INITIAL_CONDITIONS_INPUT := NOT #SWITCH_OFF_SEQUENCE_LINE_1.RUNNING AND (#iFEEDER_PLC_AUX_VALUES.i_rCarriergasActual_Line1 = 0.0) AND (#iFEEDER_PLC_AUX_VALUES.i_rDiskActual_Line1 = 0.0) AND (#iFEEDER_PLC_AUX_VALUES.i_rStirrerActual_Line1 = 0.0),
                               GAS_FLOW_ACTUAL := #iFEEDER_PLC_AUX_VALUES.i_rCarriergasActual_Line1,
                               DISK_SPEED_ACTUAL := #iFEEDER_PLC_AUX_VALUES.i_rDiskActual_Line1,
                               GAS_SETPOINT := #SWITCH_ON_SEQUENCE_LINE_1.GAS_SETPOINT,
                               DISK_SETPOINT := #SWITCH_ON_SEQUENCE_LINE_1.DISK_SETPOINT);
   END_IF;
END_REGION

REGION Network 23: SWITCH ON SEQUENCE LINE 2
   // 2#0000_0001 OPTIONS 0 BIT 0 ON SEQUENCE OPTION
   // 2#0000_0010 OPTIONS 0 BIT 1 OFF SEQUENCE OPTION
   // 2#0000_0100 OPTIONS 0 BIT 2 SPARE OPTION
   // 2#0000_1000 OPTIONS 0 BIT 3 SPARE OPTION
   // 2#0001_0000 OPTIONS 0 BIT 4 SPARE OPTION
   // 2#0010_0000 OPTIONS 0 BIT 5 SPARE OPTION
   // 2#0100_0000 OPTIONS 0 BIT 6 SPARE OPTION
   // 2#1000_0000 OPTIONS 0 BIT 7 SPARE OPTION
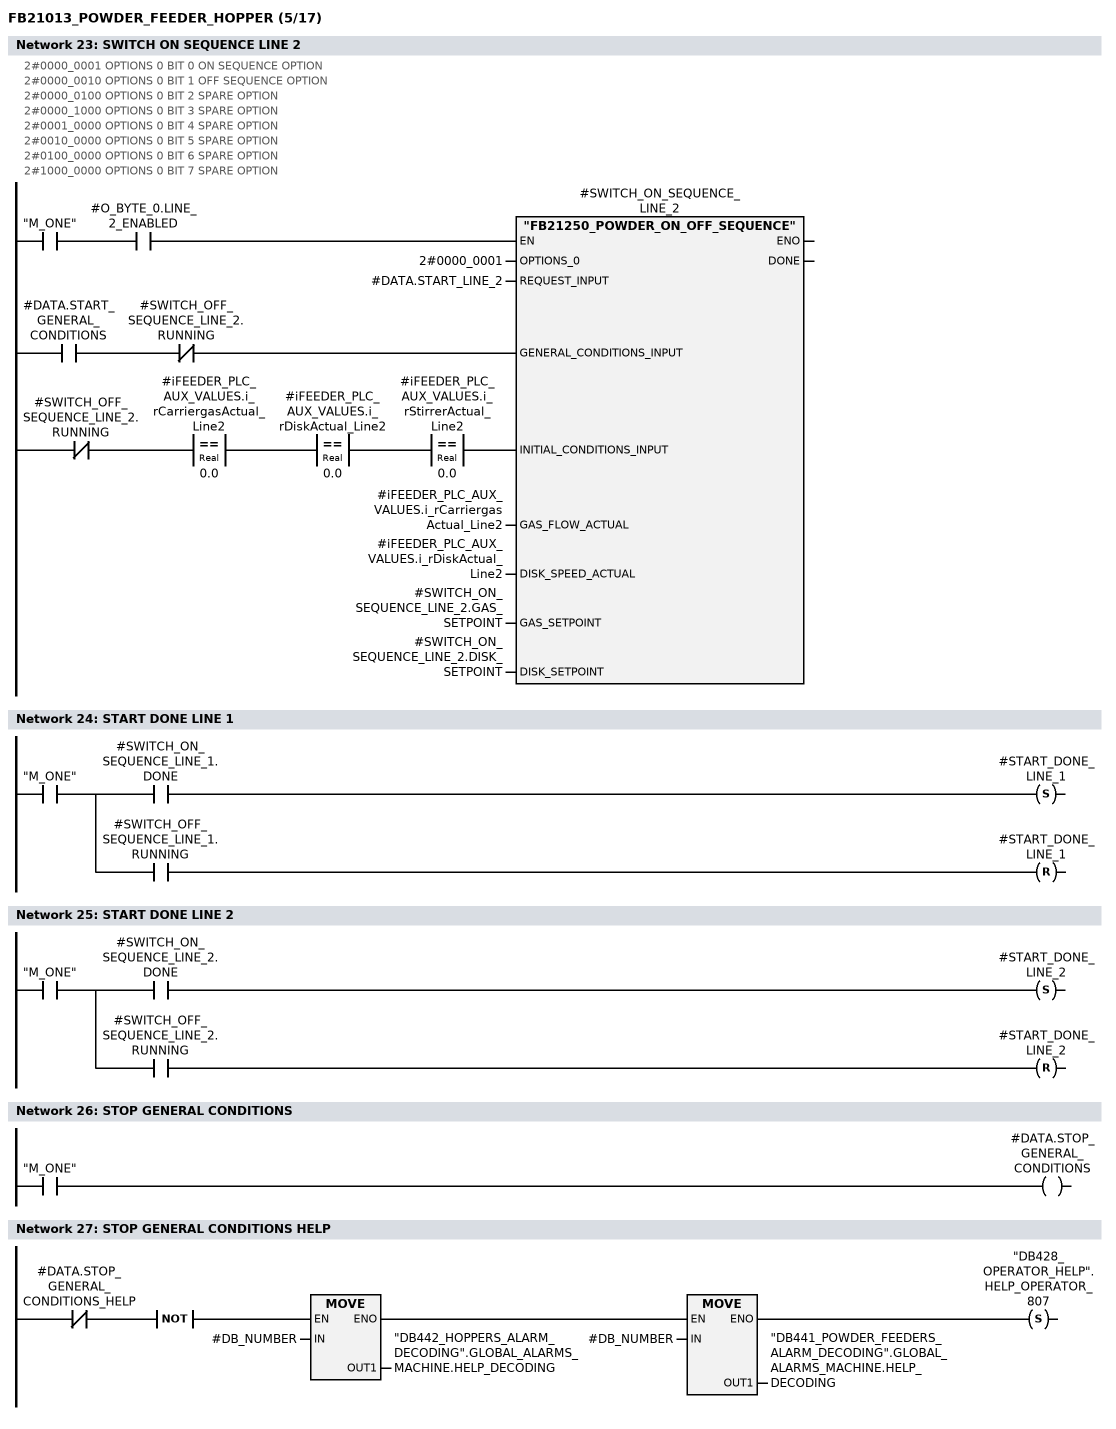
   RUNG wire#powerrail
      Contact( "M_ONE" )
      Contact( #O_BYTE_0.LINE_2_ENABLED )
      #SWITCH_ON_SEQUENCE_LINE_2(GENERAL_CONDITIONS_INPUT := wire#w1, INITIAL_CONDITIONS_INPUT := wire#w2, OPTIONS_0 := 2#0000_0001, REQUEST_INPUT := #DATA.START_LINE_2, GAS_FLOW_ACTUAL := #iFEEDER_PLC_AUX_VALUES.i_rCarriergasActual_Line2, DISK_SPEED_ACTUAL := #iFEEDER_PLC_AUX_VALUES.i_rDiskActual_Line2, GAS_SETPOINT := #SWITCH_ON_SEQUENCE_LINE_2.GAS_SETPOINT, DISK_SETPOINT := #SWITCH_ON_SEQUENCE_LINE_2.DISK_SETPOINT, DONE =>)
   END_RUNG
   RUNG wire#powerrail
      Contact( #DATA.START_GENERAL_CONDITIONS )
      I_Contact( #SWITCH_OFF_SEQUENCE_LINE_2.RUNNING )
   END_RUNG wire#w1
   RUNG wire#powerrail
      I_Contact( #SWITCH_OFF_SEQUENCE_LINE_2.RUNNING )
      { S7_Templates := "SrcType := Real" } EQ_Contact(in1 := #iFEEDER_PLC_AUX_VALUES.i_rCarriergasActual_Line2, in2 := 0.0)
      { S7_Templates := "SrcType := Real" } EQ_Contact(in1 := #iFEEDER_PLC_AUX_VALUES.i_rDiskActual_Line2, in2 := 0.0)
      { S7_Templates := "SrcType := Real" } EQ_Contact(in1 := #iFEEDER_PLC_AUX_VALUES.i_rStirrerActual_Line2, in2 := 0.0)
   END_RUNG wire#w2
   // the same network as SCL:
   IF "M_ONE" AND #O_BYTE_0.LINE_2_ENABLED THEN
       #SWITCH_ON_SEQUENCE_LINE_2(OPTIONS_0 := 2#0000_0001,   // "FB21250_POWDER_ON_OFF_SEQUENCE"
                               REQUEST_INPUT := #DATA.START_LINE_2,
                               GENERAL_CONDITIONS_INPUT := #DATA.START_GENERAL_CONDITIONS AND NOT #SWITCH_OFF_SEQUENCE_LINE_2.RUNNING,
                               INITIAL_CONDITIONS_INPUT := NOT #SWITCH_OFF_SEQUENCE_LINE_2.RUNNING AND (#iFEEDER_PLC_AUX_VALUES.i_rCarriergasActual_Line2 = 0.0) AND (#iFEEDER_PLC_AUX_VALUES.i_rDiskActual_Line2 = 0.0) AND (#iFEEDER_PLC_AUX_VALUES.i_rStirrerActual_Line2 = 0.0),
                               GAS_FLOW_ACTUAL := #iFEEDER_PLC_AUX_VALUES.i_rCarriergasActual_Line2,
                               DISK_SPEED_ACTUAL := #iFEEDER_PLC_AUX_VALUES.i_rDiskActual_Line2,
                               GAS_SETPOINT := #SWITCH_ON_SEQUENCE_LINE_2.GAS_SETPOINT,
                               DISK_SETPOINT := #SWITCH_ON_SEQUENCE_LINE_2.DISK_SETPOINT);
   END_IF;
END_REGION

REGION Network 24: START DONE LINE 1
   RUNG wire#powerrail
      Contact( "M_ONE" )
      wire#w1
      Contact( #SWITCH_ON_SEQUENCE_LINE_1.DONE )
      S_Coil( #START_DONE_LINE_1 )
   END_RUNG
   RUNG wire#w1
      Contact( #SWITCH_OFF_SEQUENCE_LINE_1.RUNNING )
      R_Coil( #START_DONE_LINE_1 )
   END_RUNG
   // the same network as SCL:
   IF "M_ONE" AND #SWITCH_ON_SEQUENCE_LINE_1.DONE THEN #START_DONE_LINE_1 := TRUE; END_IF;
   IF "M_ONE" AND #SWITCH_OFF_SEQUENCE_LINE_1.RUNNING THEN #START_DONE_LINE_1 := FALSE; END_IF;
END_REGION

REGION Network 25: START DONE LINE 2
   RUNG wire#powerrail
      Contact( "M_ONE" )
      wire#w1
      Contact( #SWITCH_ON_SEQUENCE_LINE_2.DONE )
      S_Coil( #START_DONE_LINE_2 )
   END_RUNG
   RUNG wire#w1
      Contact( #SWITCH_OFF_SEQUENCE_LINE_2.RUNNING )
      R_Coil( #START_DONE_LINE_2 )
   END_RUNG
   // the same network as SCL:
   IF "M_ONE" AND #SWITCH_ON_SEQUENCE_LINE_2.DONE THEN #START_DONE_LINE_2 := TRUE; END_IF;
   IF "M_ONE" AND #SWITCH_OFF_SEQUENCE_LINE_2.RUNNING THEN #START_DONE_LINE_2 := FALSE; END_IF;
END_REGION

REGION Network 26: STOP GENERAL CONDITIONS
   RUNG wire#powerrail
      Contact( "M_ONE" )
      Coil( #DATA.STOP_GENERAL_CONDITIONS )
   END_RUNG
   // the same network as SCL:
   #DATA.STOP_GENERAL_CONDITIONS := "M_ONE";
END_REGION

REGION Network 27: STOP GENERAL CONDITIONS HELP
   RUNG wire#powerrail
      I_Contact( #DATA.STOP_GENERAL_CONDITIONS_HELP )
      Not()
      Move(in := #DB_NUMBER, out1 => "DB442_HOPPERS_ALARM_DECODING".GLOBAL_ALARMS_MACHINE.HELP_DECODING)
      Move(in := #DB_NUMBER, out1 => "DB441_POWDER_FEEDERS_ALARM_DECODING".GLOBAL_ALARMS_MACHINE.HELP_DECODING)
      S_Coil( "DB428_OPERATOR_HELP".HELP_OPERATOR_807 )
   END_RUNG
   // the same network as SCL:
   IF NOT (NOT #DATA.STOP_GENERAL_CONDITIONS_HELP) THEN
       "DB442_HOPPERS_ALARM_DECODING".GLOBAL_ALARMS_MACHINE.HELP_DECODING := #DB_NUMBER;
       "DB441_POWDER_FEEDERS_ALARM_DECODING".GLOBAL_ALARMS_MACHINE.HELP_DECODING := #DB_NUMBER;
       "DB428_OPERATOR_HELP".HELP_OPERATOR_807 := TRUE;
   END_IF;
END_REGION

REGION Network 28: STOP INITIAL CONDITIONS LINE 1
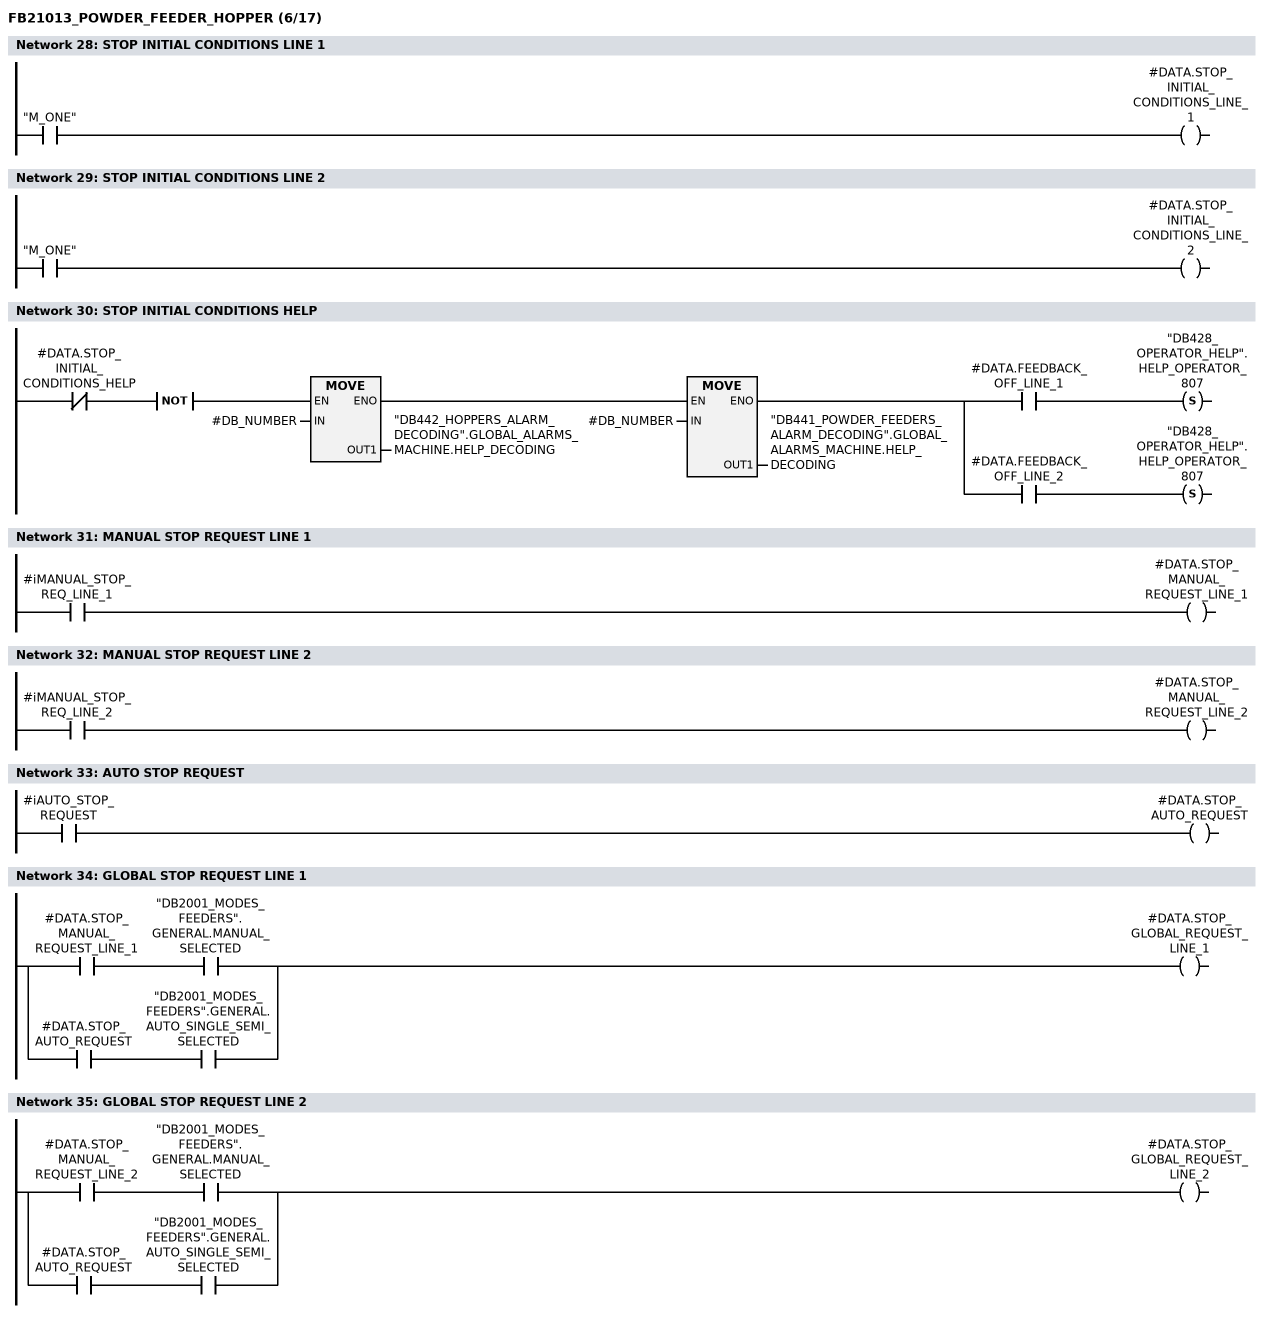
   RUNG wire#powerrail
      Contact( "M_ONE" )
      Coil( #DATA.STOP_INITIAL_CONDITIONS_LINE_1 )
   END_RUNG
   // the same network as SCL:
   #DATA.STOP_INITIAL_CONDITIONS_LINE_1 := "M_ONE";
END_REGION

REGION Network 29: STOP INITIAL CONDITIONS LINE 2
   RUNG wire#powerrail
      Contact( "M_ONE" )
      Coil( #DATA.STOP_INITIAL_CONDITIONS_LINE_2 )
   END_RUNG
   // the same network as SCL:
   #DATA.STOP_INITIAL_CONDITIONS_LINE_2 := "M_ONE";
END_REGION

REGION Network 30: STOP INITIAL CONDITIONS HELP
   RUNG wire#powerrail
      I_Contact( #DATA.STOP_INITIAL_CONDITIONS_HELP )
      Not()
      Move(in := #DB_NUMBER, out1 => "DB442_HOPPERS_ALARM_DECODING".GLOBAL_ALARMS_MACHINE.HELP_DECODING)
      Move(in := #DB_NUMBER, out1 => "DB441_POWDER_FEEDERS_ALARM_DECODING".GLOBAL_ALARMS_MACHINE.HELP_DECODING)
      wire#w1
      Contact( #DATA.FEEDBACK_OFF_LINE_1 )
      S_Coil( "DB428_OPERATOR_HELP".HELP_OPERATOR_807 )
   END_RUNG
   RUNG wire#w1
      Contact( #DATA.FEEDBACK_OFF_LINE_2 )
      S_Coil( "DB428_OPERATOR_HELP".HELP_OPERATOR_807 )
   END_RUNG
   // the same network as SCL:
   #_w1 := NOT (NOT #DATA.STOP_INITIAL_CONDITIONS_HELP);
   IF #_w1 THEN
       "DB442_HOPPERS_ALARM_DECODING".GLOBAL_ALARMS_MACHINE.HELP_DECODING := #DB_NUMBER;
       "DB441_POWDER_FEEDERS_ALARM_DECODING".GLOBAL_ALARMS_MACHINE.HELP_DECODING := #DB_NUMBER;
   END_IF;
   IF #_w1 AND #DATA.FEEDBACK_OFF_LINE_1 THEN "DB428_OPERATOR_HELP".HELP_OPERATOR_807 := TRUE; END_IF;
   IF #_w1 AND #DATA.FEEDBACK_OFF_LINE_2 THEN "DB428_OPERATOR_HELP".HELP_OPERATOR_807 := TRUE; END_IF;
END_REGION

REGION Network 31: MANUAL STOP REQUEST LINE 1
   RUNG wire#powerrail
      Contact( #iMANUAL_STOP_REQ_LINE_1 )
      Coil( #DATA.STOP_MANUAL_REQUEST_LINE_1 )
   END_RUNG
   // the same network as SCL:
   #DATA.STOP_MANUAL_REQUEST_LINE_1 := #iMANUAL_STOP_REQ_LINE_1;
END_REGION

REGION Network 32: MANUAL STOP REQUEST LINE 2
   RUNG wire#powerrail
      Contact( #iMANUAL_STOP_REQ_LINE_2 )
      Coil( #DATA.STOP_MANUAL_REQUEST_LINE_2 )
   END_RUNG
   // the same network as SCL:
   #DATA.STOP_MANUAL_REQUEST_LINE_2 := #iMANUAL_STOP_REQ_LINE_2;
END_REGION

REGION Network 33: AUTO STOP REQUEST
   RUNG wire#powerrail
      Contact( #iAUTO_STOP_REQUEST )
      Coil( #DATA.STOP_AUTO_REQUEST )
   END_RUNG
   // the same network as SCL:
   #DATA.STOP_AUTO_REQUEST := #iAUTO_STOP_REQUEST;
END_REGION

REGION Network 34: GLOBAL STOP REQUEST LINE 1
   RUNG wire#powerrail
      Contact( #DATA.STOP_MANUAL_REQUEST_LINE_1 )
      Contact( "DB2001_MODES_FEEDERS".GENERAL.MANUAL_SELECTED )
      wire#w1
      Coil( #DATA.STOP_GLOBAL_REQUEST_LINE_1 )
   END_RUNG
   RUNG wire#powerrail
      Contact( #DATA.STOP_AUTO_REQUEST )
      Contact( "DB2001_MODES_FEEDERS".GENERAL.AUTO_SINGLE_SEMI_SELECTED )
   END_RUNG wire#w1
   // the same network as SCL:
   #DATA.STOP_GLOBAL_REQUEST_LINE_1 := (#DATA.STOP_MANUAL_REQUEST_LINE_1 AND "DB2001_MODES_FEEDERS".GENERAL.MANUAL_SELECTED) OR (#DATA.STOP_AUTO_REQUEST AND "DB2001_MODES_FEEDERS".GENERAL.AUTO_SINGLE_SEMI_SELECTED);
END_REGION

REGION Network 35: GLOBAL STOP REQUEST LINE 2
   RUNG wire#powerrail
      Contact( #DATA.STOP_MANUAL_REQUEST_LINE_2 )
      Contact( "DB2001_MODES_FEEDERS".GENERAL.MANUAL_SELECTED )
      wire#w1
      Coil( #DATA.STOP_GLOBAL_REQUEST_LINE_2 )
   END_RUNG
   RUNG wire#powerrail
      Contact( #DATA.STOP_AUTO_REQUEST )
      Contact( "DB2001_MODES_FEEDERS".GENERAL.AUTO_SINGLE_SEMI_SELECTED )
   END_RUNG wire#w1
   // the same network as SCL:
   #DATA.STOP_GLOBAL_REQUEST_LINE_2 := (#DATA.STOP_MANUAL_REQUEST_LINE_2 AND "DB2001_MODES_FEEDERS".GENERAL.MANUAL_SELECTED) OR (#DATA.STOP_AUTO_REQUEST AND "DB2001_MODES_FEEDERS".GENERAL.AUTO_SINGLE_SEMI_SELECTED);
END_REGION

REGION Network 36: SWITCH OFF SEQUENCE LINE 1
   // 2#0000_0001 OPTIONS 0 BIT 0 ON SEQUENCE OPTION
   // 2#0000_0010 OPTIONS 0 BIT 1 OFF SEQUENCE OPTION
   // 2#0000_0100 OPTIONS 0 BIT 2 SPARE OPTION
   // 2#0000_1000 OPTIONS 0 BIT 3 SPARE OPTION
   // 2#0001_0000 OPTIONS 0 BIT 4 SPARE OPTION
   // 2#0010_0000 OPTIONS 0 BIT 5 SPARE OPTION
   // 2#0100_0000 OPTIONS 0 BIT 6 SPARE OPTION
   // 2#1000_0000 OPTIONS 0 BIT 7 SPARE OPTION
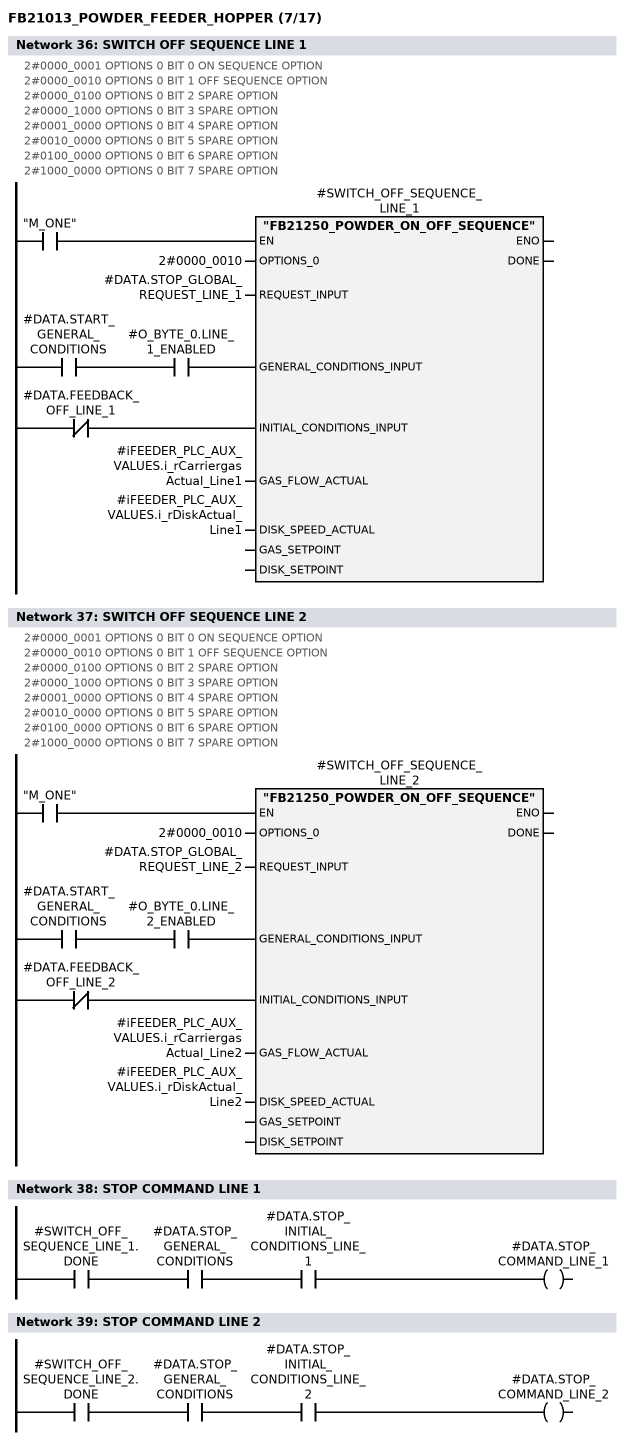
   RUNG wire#powerrail
      Contact( "M_ONE" )
      #SWITCH_OFF_SEQUENCE_LINE_1(GENERAL_CONDITIONS_INPUT := wire#w1, INITIAL_CONDITIONS_INPUT := wire#w2, OPTIONS_0 := 2#0000_0010, REQUEST_INPUT := #DATA.STOP_GLOBAL_REQUEST_LINE_1, GAS_FLOW_ACTUAL := #iFEEDER_PLC_AUX_VALUES.i_rCarriergasActual_Line1, DISK_SPEED_ACTUAL := #iFEEDER_PLC_AUX_VALUES.i_rDiskActual_Line1, GAS_SETPOINT :=, DISK_SETPOINT :=, DONE =>)
   END_RUNG
   RUNG wire#powerrail
      Contact( #DATA.START_GENERAL_CONDITIONS )
      Contact( #O_BYTE_0.LINE_1_ENABLED )
   END_RUNG wire#w1
   RUNG wire#powerrail
      I_Contact( #DATA.FEEDBACK_OFF_LINE_1 )
   END_RUNG wire#w2
   // the same network as SCL:
   IF "M_ONE" THEN
       #SWITCH_OFF_SEQUENCE_LINE_1(OPTIONS_0 := 2#0000_0010,   // "FB21250_POWDER_ON_OFF_SEQUENCE"
                               REQUEST_INPUT := #DATA.STOP_GLOBAL_REQUEST_LINE_1,
                               GENERAL_CONDITIONS_INPUT := #DATA.START_GENERAL_CONDITIONS AND #O_BYTE_0.LINE_1_ENABLED,
                               INITIAL_CONDITIONS_INPUT := NOT #DATA.FEEDBACK_OFF_LINE_1,
                               GAS_FLOW_ACTUAL := #iFEEDER_PLC_AUX_VALUES.i_rCarriergasActual_Line1,
                               DISK_SPEED_ACTUAL := #iFEEDER_PLC_AUX_VALUES.i_rDiskActual_Line1);
   END_IF;
END_REGION

REGION Network 37: SWITCH OFF SEQUENCE LINE 2
   // 2#0000_0001 OPTIONS 0 BIT 0 ON SEQUENCE OPTION
   // 2#0000_0010 OPTIONS 0 BIT 1 OFF SEQUENCE OPTION
   // 2#0000_0100 OPTIONS 0 BIT 2 SPARE OPTION
   // 2#0000_1000 OPTIONS 0 BIT 3 SPARE OPTION
   // 2#0001_0000 OPTIONS 0 BIT 4 SPARE OPTION
   // 2#0010_0000 OPTIONS 0 BIT 5 SPARE OPTION
   // 2#0100_0000 OPTIONS 0 BIT 6 SPARE OPTION
   // 2#1000_0000 OPTIONS 0 BIT 7 SPARE OPTION
   RUNG wire#powerrail
      Contact( "M_ONE" )
      #SWITCH_OFF_SEQUENCE_LINE_2(GENERAL_CONDITIONS_INPUT := wire#w1, INITIAL_CONDITIONS_INPUT := wire#w2, OPTIONS_0 := 2#0000_0010, REQUEST_INPUT := #DATA.STOP_GLOBAL_REQUEST_LINE_2, GAS_FLOW_ACTUAL := #iFEEDER_PLC_AUX_VALUES.i_rCarriergasActual_Line2, DISK_SPEED_ACTUAL := #iFEEDER_PLC_AUX_VALUES.i_rDiskActual_Line2, GAS_SETPOINT :=, DISK_SETPOINT :=, DONE =>)
   END_RUNG
   RUNG wire#powerrail
      Contact( #DATA.START_GENERAL_CONDITIONS )
      Contact( #O_BYTE_0.LINE_2_ENABLED )
   END_RUNG wire#w1
   RUNG wire#powerrail
      I_Contact( #DATA.FEEDBACK_OFF_LINE_2 )
   END_RUNG wire#w2
   // the same network as SCL:
   IF "M_ONE" THEN
       #SWITCH_OFF_SEQUENCE_LINE_2(OPTIONS_0 := 2#0000_0010,   // "FB21250_POWDER_ON_OFF_SEQUENCE"
                               REQUEST_INPUT := #DATA.STOP_GLOBAL_REQUEST_LINE_2,
                               GENERAL_CONDITIONS_INPUT := #DATA.START_GENERAL_CONDITIONS AND #O_BYTE_0.LINE_2_ENABLED,
                               INITIAL_CONDITIONS_INPUT := NOT #DATA.FEEDBACK_OFF_LINE_2,
                               GAS_FLOW_ACTUAL := #iFEEDER_PLC_AUX_VALUES.i_rCarriergasActual_Line2,
                               DISK_SPEED_ACTUAL := #iFEEDER_PLC_AUX_VALUES.i_rDiskActual_Line2);
   END_IF;
END_REGION

REGION Network 38: STOP COMMAND LINE 1
   RUNG wire#powerrail
      Contact( #SWITCH_OFF_SEQUENCE_LINE_1.DONE )
      Contact( #DATA.STOP_GENERAL_CONDITIONS )
      Contact( #DATA.STOP_INITIAL_CONDITIONS_LINE_1 )
      Coil( #DATA.STOP_COMMAND_LINE_1 )
   END_RUNG
   // the same network as SCL:
   #DATA.STOP_COMMAND_LINE_1 := #SWITCH_OFF_SEQUENCE_LINE_1.DONE AND #DATA.STOP_GENERAL_CONDITIONS AND #DATA.STOP_INITIAL_CONDITIONS_LINE_1;
END_REGION

REGION Network 39: STOP COMMAND LINE 2
   RUNG wire#powerrail
      Contact( #SWITCH_OFF_SEQUENCE_LINE_2.DONE )
      Contact( #DATA.STOP_GENERAL_CONDITIONS )
      Contact( #DATA.STOP_INITIAL_CONDITIONS_LINE_2 )
      Coil( #DATA.STOP_COMMAND_LINE_2 )
   END_RUNG
   // the same network as SCL:
   #DATA.STOP_COMMAND_LINE_2 := #SWITCH_OFF_SEQUENCE_LINE_2.DONE AND #DATA.STOP_GENERAL_CONDITIONS AND #DATA.STOP_INITIAL_CONDITIONS_LINE_2;
END_REGION

REGION Network 40: STOP LINE 1
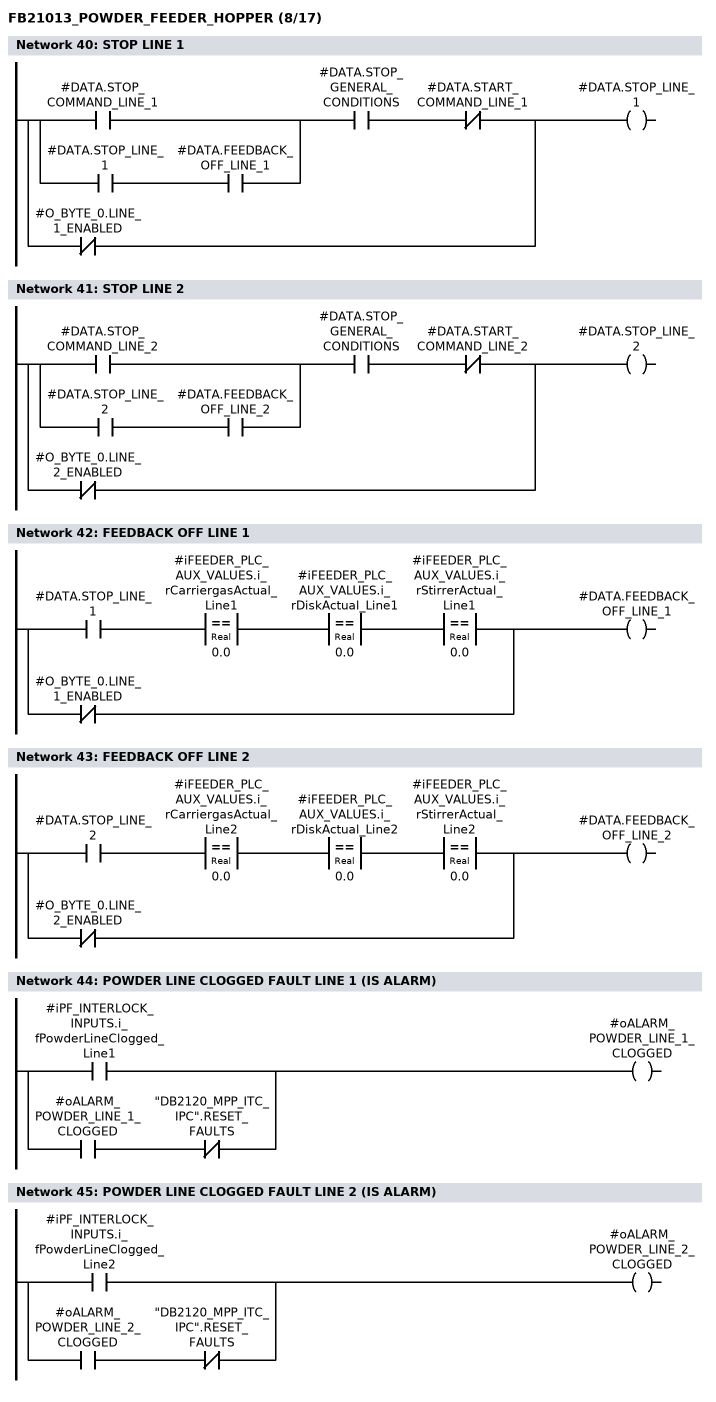
   RUNG wire#powerrail
      Contact( #DATA.STOP_COMMAND_LINE_1 )
      wire#w1
      Contact( #DATA.STOP_GENERAL_CONDITIONS )
      I_Contact( #DATA.START_COMMAND_LINE_1 )
      wire#w2
      Coil( #DATA.STOP_LINE_1 )
   END_RUNG
   RUNG wire#powerrail
      Contact( #DATA.STOP_LINE_1 )
      Contact( #DATA.FEEDBACK_OFF_LINE_1 )
   END_RUNG wire#w1
   RUNG wire#powerrail
      I_Contact( #O_BYTE_0.LINE_1_ENABLED )
   END_RUNG wire#w2
   // the same network as SCL:
   #DATA.STOP_LINE_1 := ((#DATA.STOP_COMMAND_LINE_1 OR (#DATA.STOP_LINE_1 AND #DATA.FEEDBACK_OFF_LINE_1)) AND #DATA.STOP_GENERAL_CONDITIONS AND NOT #DATA.START_COMMAND_LINE_1) OR NOT #O_BYTE_0.LINE_1_ENABLED;
END_REGION

REGION Network 41: STOP LINE 2
   RUNG wire#powerrail
      Contact( #DATA.STOP_COMMAND_LINE_2 )
      wire#w1
      Contact( #DATA.STOP_GENERAL_CONDITIONS )
      I_Contact( #DATA.START_COMMAND_LINE_2 )
      wire#w2
      Coil( #DATA.STOP_LINE_2 )
   END_RUNG
   RUNG wire#powerrail
      Contact( #DATA.STOP_LINE_2 )
      Contact( #DATA.FEEDBACK_OFF_LINE_2 )
   END_RUNG wire#w1
   RUNG wire#powerrail
      I_Contact( #O_BYTE_0.LINE_2_ENABLED )
   END_RUNG wire#w2
   // the same network as SCL:
   #DATA.STOP_LINE_2 := ((#DATA.STOP_COMMAND_LINE_2 OR (#DATA.STOP_LINE_2 AND #DATA.FEEDBACK_OFF_LINE_2)) AND #DATA.STOP_GENERAL_CONDITIONS AND NOT #DATA.START_COMMAND_LINE_2) OR NOT #O_BYTE_0.LINE_2_ENABLED;
END_REGION

REGION Network 42: FEEDBACK OFF LINE 1
   RUNG wire#powerrail
      Contact( #DATA.STOP_LINE_1 )
      { S7_Templates := "SrcType := Real" } EQ_Contact(in1 := #iFEEDER_PLC_AUX_VALUES.i_rCarriergasActual_Line1, in2 := 0.0)
      { S7_Templates := "SrcType := Real" } EQ_Contact(in1 := #iFEEDER_PLC_AUX_VALUES.i_rDiskActual_Line1, in2 := 0.0)
      { S7_Templates := "SrcType := Real" } EQ_Contact(in1 := #iFEEDER_PLC_AUX_VALUES.i_rStirrerActual_Line1, in2 := 0.0)
      wire#w1
      Coil( #DATA.FEEDBACK_OFF_LINE_1 )
   END_RUNG
   RUNG wire#powerrail
      I_Contact( #O_BYTE_0.LINE_1_ENABLED )
   END_RUNG wire#w1
   // the same network as SCL:
   #DATA.FEEDBACK_OFF_LINE_1 := (#DATA.STOP_LINE_1 AND (#iFEEDER_PLC_AUX_VALUES.i_rCarriergasActual_Line1 = 0.0) AND (#iFEEDER_PLC_AUX_VALUES.i_rDiskActual_Line1 = 0.0) AND (#iFEEDER_PLC_AUX_VALUES.i_rStirrerActual_Line1 = 0.0)) OR NOT #O_BYTE_0.LINE_1_ENABLED;
END_REGION

REGION Network 43: FEEDBACK OFF LINE 2
   RUNG wire#powerrail
      Contact( #DATA.STOP_LINE_2 )
      { S7_Templates := "SrcType := Real" } EQ_Contact(in1 := #iFEEDER_PLC_AUX_VALUES.i_rCarriergasActual_Line2, in2 := 0.0)
      { S7_Templates := "SrcType := Real" } EQ_Contact(in1 := #iFEEDER_PLC_AUX_VALUES.i_rDiskActual_Line2, in2 := 0.0)
      { S7_Templates := "SrcType := Real" } EQ_Contact(in1 := #iFEEDER_PLC_AUX_VALUES.i_rStirrerActual_Line2, in2 := 0.0)
      wire#w1
      Coil( #DATA.FEEDBACK_OFF_LINE_2 )
   END_RUNG
   RUNG wire#powerrail
      I_Contact( #O_BYTE_0.LINE_2_ENABLED )
   END_RUNG wire#w1
   // the same network as SCL:
   #DATA.FEEDBACK_OFF_LINE_2 := (#DATA.STOP_LINE_2 AND (#iFEEDER_PLC_AUX_VALUES.i_rCarriergasActual_Line2 = 0.0) AND (#iFEEDER_PLC_AUX_VALUES.i_rDiskActual_Line2 = 0.0) AND (#iFEEDER_PLC_AUX_VALUES.i_rStirrerActual_Line2 = 0.0)) OR NOT #O_BYTE_0.LINE_2_ENABLED;
END_REGION

REGION Network 44: POWDER LINE CLOGGED FAULT LINE 1 (IS ALARM)
   RUNG wire#powerrail
      Contact( #iPF_INTERLOCK_INPUTS.i_fPowderLineClogged_Line1 )
      wire#w1
      Coil( #oALARM_POWDER_LINE_1_CLOGGED )
   END_RUNG
   RUNG wire#powerrail
      Contact( #oALARM_POWDER_LINE_1_CLOGGED )
      I_Contact( "DB2120_MPP_ITC_IPC".RESET_FAULTS )
   END_RUNG wire#w1
   // the same network as SCL:
   #oALARM_POWDER_LINE_1_CLOGGED := #iPF_INTERLOCK_INPUTS.i_fPowderLineClogged_Line1 OR (#oALARM_POWDER_LINE_1_CLOGGED AND NOT "DB2120_MPP_ITC_IPC".RESET_FAULTS);
END_REGION

REGION Network 45: POWDER LINE CLOGGED FAULT LINE 2 (IS ALARM)
   RUNG wire#powerrail
      Contact( #iPF_INTERLOCK_INPUTS.i_fPowderLineClogged_Line2 )
      wire#w1
      Coil( #oALARM_POWDER_LINE_2_CLOGGED )
   END_RUNG
   RUNG wire#powerrail
      Contact( #oALARM_POWDER_LINE_2_CLOGGED )
      I_Contact( "DB2120_MPP_ITC_IPC".RESET_FAULTS )
   END_RUNG wire#w1
   // the same network as SCL:
   #oALARM_POWDER_LINE_2_CLOGGED := #iPF_INTERLOCK_INPUTS.i_fPowderLineClogged_Line2 OR (#oALARM_POWDER_LINE_2_CLOGGED AND NOT "DB2120_MPP_ITC_IPC".RESET_FAULTS);
END_REGION

REGION Network 46: CARRIER GAS FLOW BELOW LOW LIMIT FAULT LINE 1 (IS ALARM)
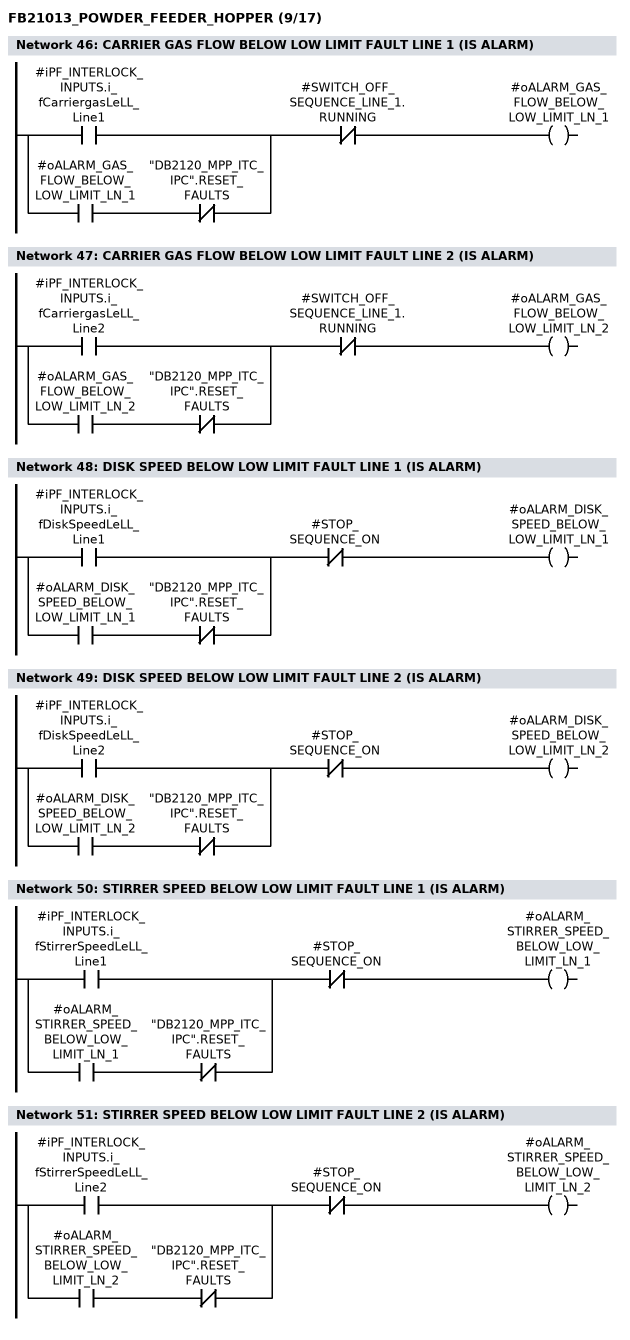
   RUNG wire#powerrail
      Contact( #iPF_INTERLOCK_INPUTS.i_fCarriergasLeLL_Line1 )
      wire#w1
      I_Contact( #SWITCH_OFF_SEQUENCE_LINE_1.RUNNING )
      Coil( #oALARM_GAS_FLOW_BELOW_LOW_LIMIT_LN_1 )
   END_RUNG
   RUNG wire#powerrail
      Contact( #oALARM_GAS_FLOW_BELOW_LOW_LIMIT_LN_1 )
      I_Contact( "DB2120_MPP_ITC_IPC".RESET_FAULTS )
   END_RUNG wire#w1
   // the same network as SCL:
   #oALARM_GAS_FLOW_BELOW_LOW_LIMIT_LN_1 := (#iPF_INTERLOCK_INPUTS.i_fCarriergasLeLL_Line1 OR (#oALARM_GAS_FLOW_BELOW_LOW_LIMIT_LN_1 AND NOT "DB2120_MPP_ITC_IPC".RESET_FAULTS)) AND NOT #SWITCH_OFF_SEQUENCE_LINE_1.RUNNING;
END_REGION

REGION Network 47: CARRIER GAS FLOW BELOW LOW LIMIT FAULT LINE 2 (IS ALARM)
   RUNG wire#powerrail
      Contact( #iPF_INTERLOCK_INPUTS.i_fCarriergasLeLL_Line2 )
      wire#w1
      I_Contact( #SWITCH_OFF_SEQUENCE_LINE_1.RUNNING )
      Coil( #oALARM_GAS_FLOW_BELOW_LOW_LIMIT_LN_2 )
   END_RUNG
   RUNG wire#powerrail
      Contact( #oALARM_GAS_FLOW_BELOW_LOW_LIMIT_LN_2 )
      I_Contact( "DB2120_MPP_ITC_IPC".RESET_FAULTS )
   END_RUNG wire#w1
   // the same network as SCL:
   #oALARM_GAS_FLOW_BELOW_LOW_LIMIT_LN_2 := (#iPF_INTERLOCK_INPUTS.i_fCarriergasLeLL_Line2 OR (#oALARM_GAS_FLOW_BELOW_LOW_LIMIT_LN_2 AND NOT "DB2120_MPP_ITC_IPC".RESET_FAULTS)) AND NOT #SWITCH_OFF_SEQUENCE_LINE_1.RUNNING;
END_REGION

REGION Network 48: DISK SPEED BELOW LOW LIMIT FAULT LINE 1 (IS ALARM)
   RUNG wire#powerrail
      Contact( #iPF_INTERLOCK_INPUTS.i_fDiskSpeedLeLL_Line1 )
      wire#w1
      I_Contact( #STOP_SEQUENCE_ON )
      Coil( #oALARM_DISK_SPEED_BELOW_LOW_LIMIT_LN_1 )
   END_RUNG
   RUNG wire#powerrail
      Contact( #oALARM_DISK_SPEED_BELOW_LOW_LIMIT_LN_1 )
      I_Contact( "DB2120_MPP_ITC_IPC".RESET_FAULTS )
   END_RUNG wire#w1
   // the same network as SCL:
   #oALARM_DISK_SPEED_BELOW_LOW_LIMIT_LN_1 := (#iPF_INTERLOCK_INPUTS.i_fDiskSpeedLeLL_Line1 OR (#oALARM_DISK_SPEED_BELOW_LOW_LIMIT_LN_1 AND NOT "DB2120_MPP_ITC_IPC".RESET_FAULTS)) AND NOT #STOP_SEQUENCE_ON;
END_REGION

REGION Network 49: DISK SPEED BELOW LOW LIMIT FAULT LINE 2 (IS ALARM)
   RUNG wire#powerrail
      Contact( #iPF_INTERLOCK_INPUTS.i_fDiskSpeedLeLL_Line2 )
      wire#w1
      I_Contact( #STOP_SEQUENCE_ON )
      Coil( #oALARM_DISK_SPEED_BELOW_LOW_LIMIT_LN_2 )
   END_RUNG
   RUNG wire#powerrail
      Contact( #oALARM_DISK_SPEED_BELOW_LOW_LIMIT_LN_2 )
      I_Contact( "DB2120_MPP_ITC_IPC".RESET_FAULTS )
   END_RUNG wire#w1
   // the same network as SCL:
   #oALARM_DISK_SPEED_BELOW_LOW_LIMIT_LN_2 := (#iPF_INTERLOCK_INPUTS.i_fDiskSpeedLeLL_Line2 OR (#oALARM_DISK_SPEED_BELOW_LOW_LIMIT_LN_2 AND NOT "DB2120_MPP_ITC_IPC".RESET_FAULTS)) AND NOT #STOP_SEQUENCE_ON;
END_REGION

REGION Network 50: STIRRER SPEED BELOW LOW LIMIT FAULT LINE 1 (IS ALARM)
   RUNG wire#powerrail
      Contact( #iPF_INTERLOCK_INPUTS.i_fStirrerSpeedLeLL_Line1 )
      wire#w1
      I_Contact( #STOP_SEQUENCE_ON )
      Coil( #oALARM_STIRRER_SPEED_BELOW_LOW_LIMIT_LN_1 )
   END_RUNG
   RUNG wire#powerrail
      Contact( #oALARM_STIRRER_SPEED_BELOW_LOW_LIMIT_LN_1 )
      I_Contact( "DB2120_MPP_ITC_IPC".RESET_FAULTS )
   END_RUNG wire#w1
   // the same network as SCL:
   #oALARM_STIRRER_SPEED_BELOW_LOW_LIMIT_LN_1 := (#iPF_INTERLOCK_INPUTS.i_fStirrerSpeedLeLL_Line1 OR (#oALARM_STIRRER_SPEED_BELOW_LOW_LIMIT_LN_1 AND NOT "DB2120_MPP_ITC_IPC".RESET_FAULTS)) AND NOT #STOP_SEQUENCE_ON;
END_REGION

REGION Network 51: STIRRER SPEED BELOW LOW LIMIT FAULT LINE 2 (IS ALARM)
   RUNG wire#powerrail
      Contact( #iPF_INTERLOCK_INPUTS.i_fStirrerSpeedLeLL_Line2 )
      wire#w1
      I_Contact( #STOP_SEQUENCE_ON )
      Coil( #oALARM_STIRRER_SPEED_BELOW_LOW_LIMIT_LN_2 )
   END_RUNG
   RUNG wire#powerrail
      Contact( #oALARM_STIRRER_SPEED_BELOW_LOW_LIMIT_LN_2 )
      I_Contact( "DB2120_MPP_ITC_IPC".RESET_FAULTS )
   END_RUNG wire#w1
   // the same network as SCL:
   #oALARM_STIRRER_SPEED_BELOW_LOW_LIMIT_LN_2 := (#iPF_INTERLOCK_INPUTS.i_fStirrerSpeedLeLL_Line2 OR (#oALARM_STIRRER_SPEED_BELOW_LOW_LIMIT_LN_2 AND NOT "DB2120_MPP_ITC_IPC".RESET_FAULTS)) AND NOT #STOP_SEQUENCE_ON;
END_REGION

REGION Network 52: CARRIER GAS FLOW ABOVE HIGH LIMIT FAULT LINE 1 (IS ALARM)
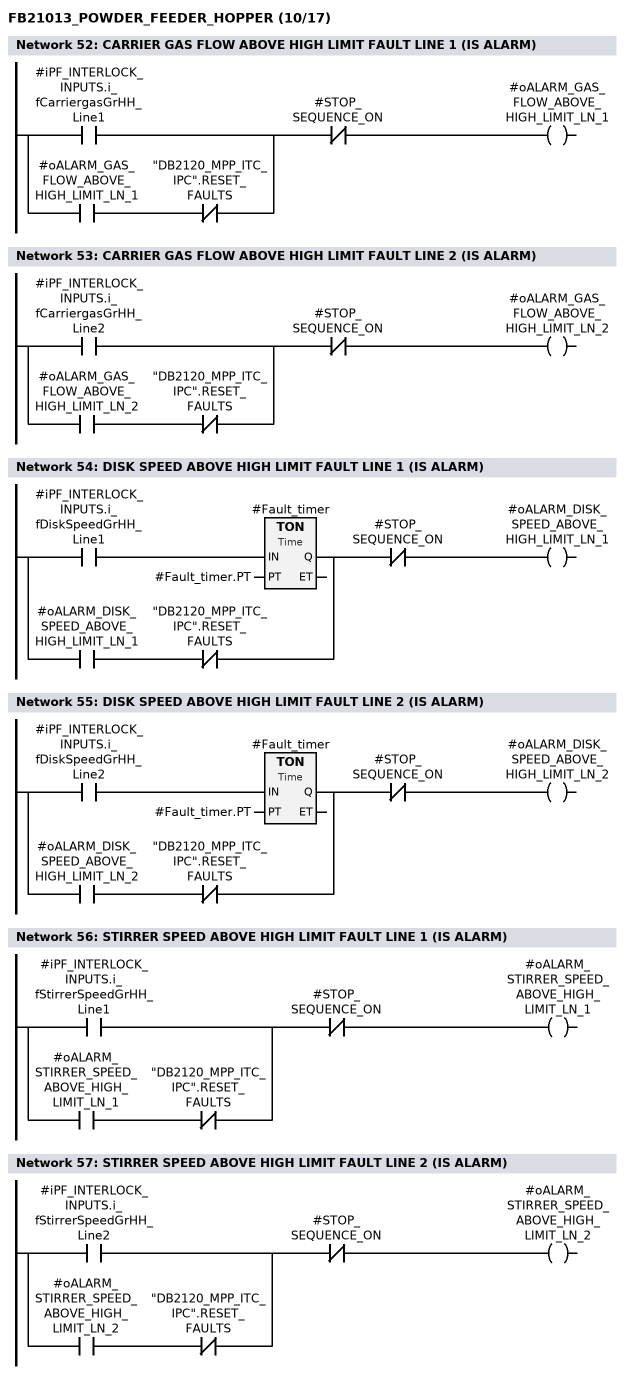
   RUNG wire#powerrail
      Contact( #iPF_INTERLOCK_INPUTS.i_fCarriergasGrHH_Line1 )
      wire#w1
      I_Contact( #STOP_SEQUENCE_ON )
      Coil( #oALARM_GAS_FLOW_ABOVE_HIGH_LIMIT_LN_1 )
   END_RUNG
   RUNG wire#powerrail
      Contact( #oALARM_GAS_FLOW_ABOVE_HIGH_LIMIT_LN_1 )
      I_Contact( "DB2120_MPP_ITC_IPC".RESET_FAULTS )
   END_RUNG wire#w1
   // the same network as SCL:
   #oALARM_GAS_FLOW_ABOVE_HIGH_LIMIT_LN_1 := (#iPF_INTERLOCK_INPUTS.i_fCarriergasGrHH_Line1 OR (#oALARM_GAS_FLOW_ABOVE_HIGH_LIMIT_LN_1 AND NOT "DB2120_MPP_ITC_IPC".RESET_FAULTS)) AND NOT #STOP_SEQUENCE_ON;
END_REGION

REGION Network 53: CARRIER GAS FLOW ABOVE HIGH LIMIT FAULT LINE 2 (IS ALARM)
   RUNG wire#powerrail
      Contact( #iPF_INTERLOCK_INPUTS.i_fCarriergasGrHH_Line2 )
      wire#w1
      I_Contact( #STOP_SEQUENCE_ON )
      Coil( #oALARM_GAS_FLOW_ABOVE_HIGH_LIMIT_LN_2 )
   END_RUNG
   RUNG wire#powerrail
      Contact( #oALARM_GAS_FLOW_ABOVE_HIGH_LIMIT_LN_2 )
      I_Contact( "DB2120_MPP_ITC_IPC".RESET_FAULTS )
   END_RUNG wire#w1
   // the same network as SCL:
   #oALARM_GAS_FLOW_ABOVE_HIGH_LIMIT_LN_2 := (#iPF_INTERLOCK_INPUTS.i_fCarriergasGrHH_Line2 OR (#oALARM_GAS_FLOW_ABOVE_HIGH_LIMIT_LN_2 AND NOT "DB2120_MPP_ITC_IPC".RESET_FAULTS)) AND NOT #STOP_SEQUENCE_ON;
END_REGION

REGION Network 54: DISK SPEED ABOVE HIGH LIMIT FAULT LINE 1 (IS ALARM)
   RUNG wire#powerrail
      Contact( #iPF_INTERLOCK_INPUTS.i_fDiskSpeedGrHH_Line1 )
      { S7_Templates := "time_type := Time" } #Fault_timer.TON(pt := #Fault_timer.PT, et =>)
      wire#w1
      I_Contact( #STOP_SEQUENCE_ON )
      Coil( #oALARM_DISK_SPEED_ABOVE_HIGH_LIMIT_LN_1 )
   END_RUNG
   RUNG wire#powerrail
      Contact( #oALARM_DISK_SPEED_ABOVE_HIGH_LIMIT_LN_1 )
      I_Contact( "DB2120_MPP_ITC_IPC".RESET_FAULTS )
   END_RUNG wire#w1
   // the same network as SCL:
   #Fault_timer(IN := #iPF_INTERLOCK_INPUTS.i_fDiskSpeedGrHH_Line1, PT := #Fault_timer.PT);   // TON
   #oALARM_DISK_SPEED_ABOVE_HIGH_LIMIT_LN_1 := (#Fault_timer.Q OR (#oALARM_DISK_SPEED_ABOVE_HIGH_LIMIT_LN_1 AND NOT "DB2120_MPP_ITC_IPC".RESET_FAULTS)) AND NOT #STOP_SEQUENCE_ON;
END_REGION

REGION Network 55: DISK SPEED ABOVE HIGH LIMIT FAULT LINE 2 (IS ALARM)
   RUNG wire#powerrail
      Contact( #iPF_INTERLOCK_INPUTS.i_fDiskSpeedGrHH_Line2 )
      { S7_Templates := "time_type := Time" } #Fault_timer.TON(pt := #Fault_timer.PT, et =>)
      wire#w1
      I_Contact( #STOP_SEQUENCE_ON )
      Coil( #oALARM_DISK_SPEED_ABOVE_HIGH_LIMIT_LN_2 )
   END_RUNG
   RUNG wire#powerrail
      Contact( #oALARM_DISK_SPEED_ABOVE_HIGH_LIMIT_LN_2 )
      I_Contact( "DB2120_MPP_ITC_IPC".RESET_FAULTS )
   END_RUNG wire#w1
   // the same network as SCL:
   #Fault_timer(IN := #iPF_INTERLOCK_INPUTS.i_fDiskSpeedGrHH_Line2, PT := #Fault_timer.PT);   // TON
   #oALARM_DISK_SPEED_ABOVE_HIGH_LIMIT_LN_2 := (#Fault_timer.Q OR (#oALARM_DISK_SPEED_ABOVE_HIGH_LIMIT_LN_2 AND NOT "DB2120_MPP_ITC_IPC".RESET_FAULTS)) AND NOT #STOP_SEQUENCE_ON;
END_REGION

REGION Network 56: STIRRER SPEED ABOVE HIGH LIMIT FAULT LINE 1 (IS ALARM)
   RUNG wire#powerrail
      Contact( #iPF_INTERLOCK_INPUTS.i_fStirrerSpeedGrHH_Line1 )
      wire#w1
      I_Contact( #STOP_SEQUENCE_ON )
      Coil( #oALARM_STIRRER_SPEED_ABOVE_HIGH_LIMIT_LN_1 )
   END_RUNG
   RUNG wire#powerrail
      Contact( #oALARM_STIRRER_SPEED_ABOVE_HIGH_LIMIT_LN_1 )
      I_Contact( "DB2120_MPP_ITC_IPC".RESET_FAULTS )
   END_RUNG wire#w1
   // the same network as SCL:
   #oALARM_STIRRER_SPEED_ABOVE_HIGH_LIMIT_LN_1 := (#iPF_INTERLOCK_INPUTS.i_fStirrerSpeedGrHH_Line1 OR (#oALARM_STIRRER_SPEED_ABOVE_HIGH_LIMIT_LN_1 AND NOT "DB2120_MPP_ITC_IPC".RESET_FAULTS)) AND NOT #STOP_SEQUENCE_ON;
END_REGION

REGION Network 57: STIRRER SPEED ABOVE HIGH LIMIT FAULT LINE 2 (IS ALARM)
   RUNG wire#powerrail
      Contact( #iPF_INTERLOCK_INPUTS.i_fStirrerSpeedGrHH_Line2 )
      wire#w1
      I_Contact( #STOP_SEQUENCE_ON )
      Coil( #oALARM_STIRRER_SPEED_ABOVE_HIGH_LIMIT_LN_2 )
   END_RUNG
   RUNG wire#powerrail
      Contact( #oALARM_STIRRER_SPEED_ABOVE_HIGH_LIMIT_LN_2 )
      I_Contact( "DB2120_MPP_ITC_IPC".RESET_FAULTS )
   END_RUNG wire#w1
   // the same network as SCL:
   #oALARM_STIRRER_SPEED_ABOVE_HIGH_LIMIT_LN_2 := (#iPF_INTERLOCK_INPUTS.i_fStirrerSpeedGrHH_Line2 OR (#oALARM_STIRRER_SPEED_ABOVE_HIGH_LIMIT_LN_2 AND NOT "DB2120_MPP_ITC_IPC".RESET_FAULTS)) AND NOT #STOP_SEQUENCE_ON;
END_REGION

REGION Network 58: CARRIERGAS INLET PRESSURE TOO LOW LINE LINE 1
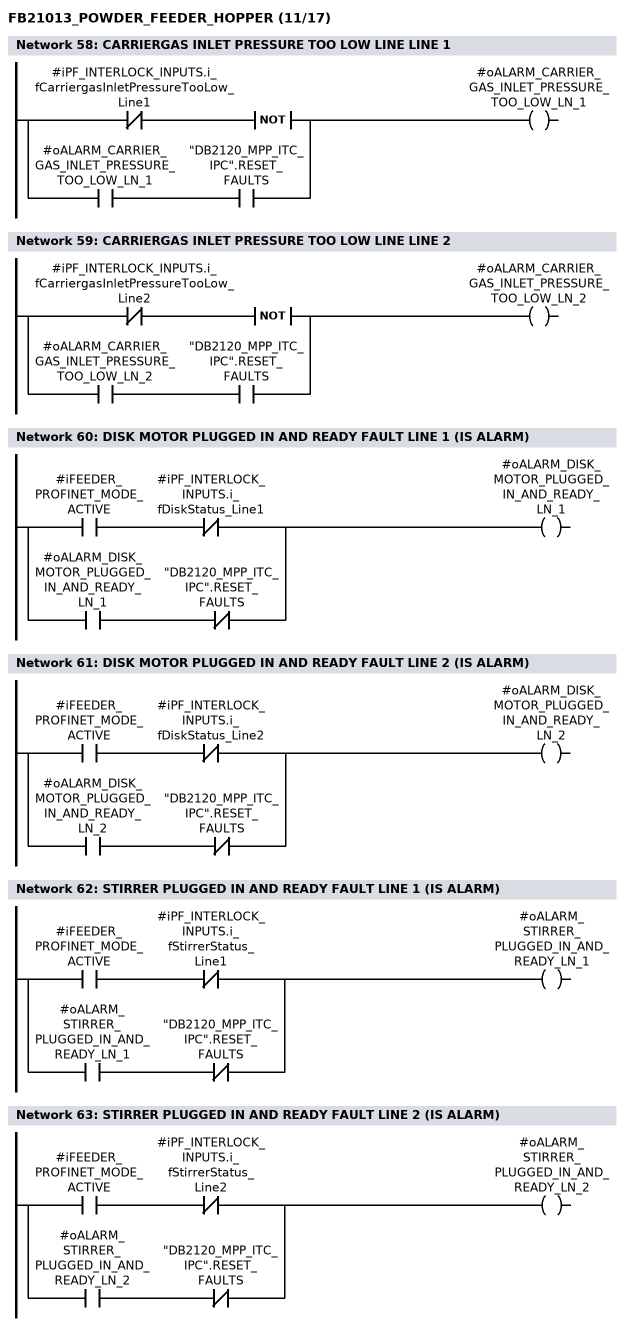
   RUNG wire#powerrail
      I_Contact( #iPF_INTERLOCK_INPUTS.i_fCarriergasInletPressureTooLow_Line1 )
      Not()
      wire#w1
      Coil( #oALARM_CARRIER_GAS_INLET_PRESSURE_TOO_LOW_LN_1 )
   END_RUNG
   RUNG wire#powerrail
      Contact( #oALARM_CARRIER_GAS_INLET_PRESSURE_TOO_LOW_LN_1 )
      Contact( "DB2120_MPP_ITC_IPC".RESET_FAULTS )
   END_RUNG wire#w1
   // the same network as SCL:
   #oALARM_CARRIER_GAS_INLET_PRESSURE_TOO_LOW_LN_1 := NOT (NOT #iPF_INTERLOCK_INPUTS.i_fCarriergasInletPressureTooLow_Line1) OR (#oALARM_CARRIER_GAS_INLET_PRESSURE_TOO_LOW_LN_1 AND "DB2120_MPP_ITC_IPC".RESET_FAULTS);
END_REGION

REGION Network 59: CARRIERGAS INLET PRESSURE TOO LOW LINE LINE 2
   RUNG wire#powerrail
      I_Contact( #iPF_INTERLOCK_INPUTS.i_fCarriergasInletPressureTooLow_Line2 )
      Not()
      wire#w1
      Coil( #oALARM_CARRIER_GAS_INLET_PRESSURE_TOO_LOW_LN_2 )
   END_RUNG
   RUNG wire#powerrail
      Contact( #oALARM_CARRIER_GAS_INLET_PRESSURE_TOO_LOW_LN_2 )
      Contact( "DB2120_MPP_ITC_IPC".RESET_FAULTS )
   END_RUNG wire#w1
   // the same network as SCL:
   #oALARM_CARRIER_GAS_INLET_PRESSURE_TOO_LOW_LN_2 := NOT (NOT #iPF_INTERLOCK_INPUTS.i_fCarriergasInletPressureTooLow_Line2) OR (#oALARM_CARRIER_GAS_INLET_PRESSURE_TOO_LOW_LN_2 AND "DB2120_MPP_ITC_IPC".RESET_FAULTS);
END_REGION

REGION Network 60: DISK MOTOR PLUGGED IN AND READY FAULT LINE 1 (IS ALARM)
   RUNG wire#powerrail
      Contact( #iFEEDER_PROFINET_MODE_ACTIVE )
      I_Contact( #iPF_INTERLOCK_INPUTS.i_fDiskStatus_Line1 )
      wire#w1
      Coil( #oALARM_DISK_MOTOR_PLUGGED_IN_AND_READY_LN_1 )
   END_RUNG
   RUNG wire#powerrail
      Contact( #oALARM_DISK_MOTOR_PLUGGED_IN_AND_READY_LN_1 )
      I_Contact( "DB2120_MPP_ITC_IPC".RESET_FAULTS )
   END_RUNG wire#w1
   // the same network as SCL:
   #oALARM_DISK_MOTOR_PLUGGED_IN_AND_READY_LN_1 := (#iFEEDER_PROFINET_MODE_ACTIVE AND NOT #iPF_INTERLOCK_INPUTS.i_fDiskStatus_Line1) OR (#oALARM_DISK_MOTOR_PLUGGED_IN_AND_READY_LN_1 AND NOT "DB2120_MPP_ITC_IPC".RESET_FAULTS);
END_REGION

REGION Network 61: DISK MOTOR PLUGGED IN AND READY FAULT LINE 2 (IS ALARM)
   RUNG wire#powerrail
      Contact( #iFEEDER_PROFINET_MODE_ACTIVE )
      I_Contact( #iPF_INTERLOCK_INPUTS.i_fDiskStatus_Line2 )
      wire#w1
      Coil( #oALARM_DISK_MOTOR_PLUGGED_IN_AND_READY_LN_2 )
   END_RUNG
   RUNG wire#powerrail
      Contact( #oALARM_DISK_MOTOR_PLUGGED_IN_AND_READY_LN_2 )
      I_Contact( "DB2120_MPP_ITC_IPC".RESET_FAULTS )
   END_RUNG wire#w1
   // the same network as SCL:
   #oALARM_DISK_MOTOR_PLUGGED_IN_AND_READY_LN_2 := (#iFEEDER_PROFINET_MODE_ACTIVE AND NOT #iPF_INTERLOCK_INPUTS.i_fDiskStatus_Line2) OR (#oALARM_DISK_MOTOR_PLUGGED_IN_AND_READY_LN_2 AND NOT "DB2120_MPP_ITC_IPC".RESET_FAULTS);
END_REGION

REGION Network 62: STIRRER PLUGGED IN AND READY FAULT LINE 1 (IS ALARM)
   RUNG wire#powerrail
      Contact( #iFEEDER_PROFINET_MODE_ACTIVE )
      I_Contact( #iPF_INTERLOCK_INPUTS.i_fStirrerStatus_Line1 )
      wire#w1
      Coil( #oALARM_STIRRER_PLUGGED_IN_AND_READY_LN_1 )
   END_RUNG
   RUNG wire#powerrail
      Contact( #oALARM_STIRRER_PLUGGED_IN_AND_READY_LN_1 )
      I_Contact( "DB2120_MPP_ITC_IPC".RESET_FAULTS )
   END_RUNG wire#w1
   // the same network as SCL:
   #oALARM_STIRRER_PLUGGED_IN_AND_READY_LN_1 := (#iFEEDER_PROFINET_MODE_ACTIVE AND NOT #iPF_INTERLOCK_INPUTS.i_fStirrerStatus_Line1) OR (#oALARM_STIRRER_PLUGGED_IN_AND_READY_LN_1 AND NOT "DB2120_MPP_ITC_IPC".RESET_FAULTS);
END_REGION

REGION Network 63: STIRRER PLUGGED IN AND READY FAULT LINE 2 (IS ALARM)
   RUNG wire#powerrail
      Contact( #iFEEDER_PROFINET_MODE_ACTIVE )
      I_Contact( #iPF_INTERLOCK_INPUTS.i_fStirrerStatus_Line2 )
      wire#w1
      Coil( #oALARM_STIRRER_PLUGGED_IN_AND_READY_LN_2 )
   END_RUNG
   RUNG wire#powerrail
      Contact( #oALARM_STIRRER_PLUGGED_IN_AND_READY_LN_2 )
      I_Contact( "DB2120_MPP_ITC_IPC".RESET_FAULTS )
   END_RUNG wire#w1
   // the same network as SCL:
   #oALARM_STIRRER_PLUGGED_IN_AND_READY_LN_2 := (#iFEEDER_PROFINET_MODE_ACTIVE AND NOT #iPF_INTERLOCK_INPUTS.i_fStirrerStatus_Line2) OR (#oALARM_STIRRER_PLUGGED_IN_AND_READY_LN_2 AND NOT "DB2120_MPP_ITC_IPC".RESET_FAULTS);
END_REGION

REGION Network 64: COMMUNICATION RUNNING FAULT LINE 1 (IS ALARM)
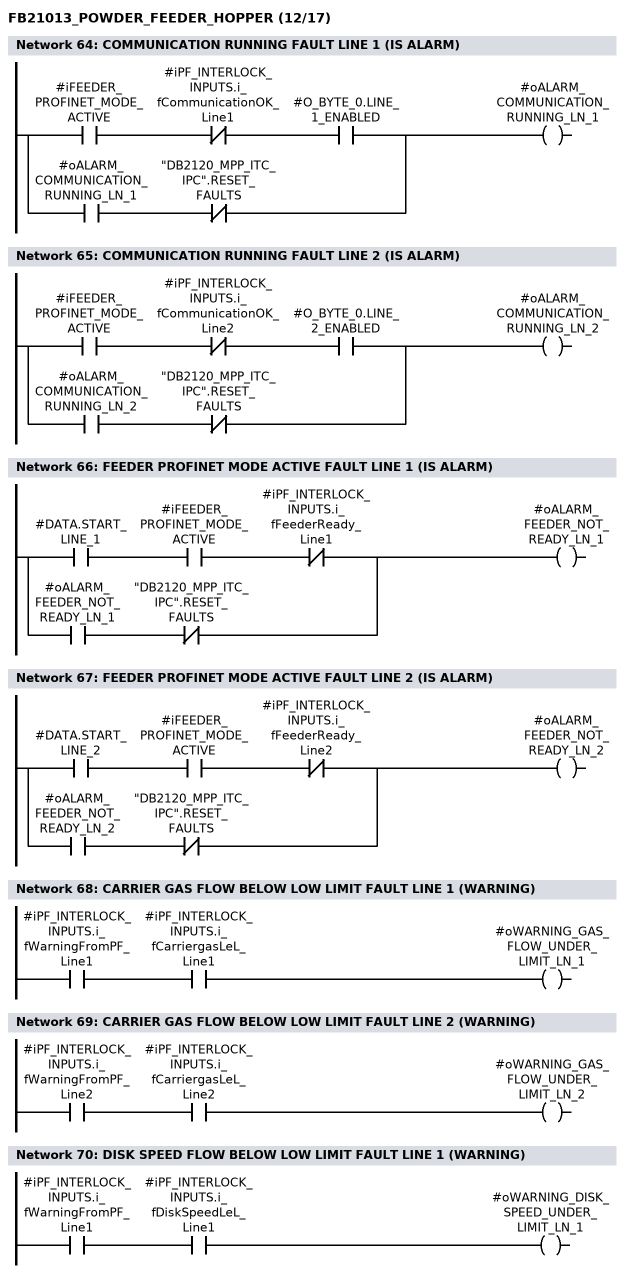
   RUNG wire#powerrail
      Contact( #iFEEDER_PROFINET_MODE_ACTIVE )
      I_Contact( #iPF_INTERLOCK_INPUTS.i_fCommunicationOK_Line1 )
      Contact( #O_BYTE_0.LINE_1_ENABLED )
      wire#w1
      Coil( #oALARM_COMMUNICATION_RUNNING_LN_1 )
   END_RUNG
   RUNG wire#powerrail
      Contact( #oALARM_COMMUNICATION_RUNNING_LN_1 )
      I_Contact( "DB2120_MPP_ITC_IPC".RESET_FAULTS )
   END_RUNG wire#w1
   // the same network as SCL:
   #oALARM_COMMUNICATION_RUNNING_LN_1 := (#iFEEDER_PROFINET_MODE_ACTIVE AND NOT #iPF_INTERLOCK_INPUTS.i_fCommunicationOK_Line1 AND #O_BYTE_0.LINE_1_ENABLED) OR (#oALARM_COMMUNICATION_RUNNING_LN_1 AND NOT "DB2120_MPP_ITC_IPC".RESET_FAULTS);
END_REGION

REGION Network 65: COMMUNICATION RUNNING FAULT LINE 2 (IS ALARM)
   RUNG wire#powerrail
      Contact( #iFEEDER_PROFINET_MODE_ACTIVE )
      I_Contact( #iPF_INTERLOCK_INPUTS.i_fCommunicationOK_Line2 )
      Contact( #O_BYTE_0.LINE_2_ENABLED )
      wire#w1
      Coil( #oALARM_COMMUNICATION_RUNNING_LN_2 )
   END_RUNG
   RUNG wire#powerrail
      Contact( #oALARM_COMMUNICATION_RUNNING_LN_2 )
      I_Contact( "DB2120_MPP_ITC_IPC".RESET_FAULTS )
   END_RUNG wire#w1
   // the same network as SCL:
   #oALARM_COMMUNICATION_RUNNING_LN_2 := (#iFEEDER_PROFINET_MODE_ACTIVE AND NOT #iPF_INTERLOCK_INPUTS.i_fCommunicationOK_Line2 AND #O_BYTE_0.LINE_2_ENABLED) OR (#oALARM_COMMUNICATION_RUNNING_LN_2 AND NOT "DB2120_MPP_ITC_IPC".RESET_FAULTS);
END_REGION

REGION Network 66: FEEDER PROFINET MODE ACTIVE FAULT LINE 1 (IS ALARM)
   RUNG wire#powerrail
      Contact( #DATA.START_LINE_1 )
      Contact( #iFEEDER_PROFINET_MODE_ACTIVE )
      I_Contact( #iPF_INTERLOCK_INPUTS.i_fFeederReady_Line1 )
      wire#w1
      Coil( #oALARM_FEEDER_NOT_READY_LN_1 )
   END_RUNG
   RUNG wire#powerrail
      Contact( #oALARM_FEEDER_NOT_READY_LN_1 )
      I_Contact( "DB2120_MPP_ITC_IPC".RESET_FAULTS )
   END_RUNG wire#w1
   // the same network as SCL:
   #oALARM_FEEDER_NOT_READY_LN_1 := (#DATA.START_LINE_1 AND #iFEEDER_PROFINET_MODE_ACTIVE AND NOT #iPF_INTERLOCK_INPUTS.i_fFeederReady_Line1) OR (#oALARM_FEEDER_NOT_READY_LN_1 AND NOT "DB2120_MPP_ITC_IPC".RESET_FAULTS);
END_REGION

REGION Network 67: FEEDER PROFINET MODE ACTIVE FAULT LINE 2 (IS ALARM)
   RUNG wire#powerrail
      Contact( #DATA.START_LINE_2 )
      Contact( #iFEEDER_PROFINET_MODE_ACTIVE )
      I_Contact( #iPF_INTERLOCK_INPUTS.i_fFeederReady_Line2 )
      wire#w1
      Coil( #oALARM_FEEDER_NOT_READY_LN_2 )
   END_RUNG
   RUNG wire#powerrail
      Contact( #oALARM_FEEDER_NOT_READY_LN_2 )
      I_Contact( "DB2120_MPP_ITC_IPC".RESET_FAULTS )
   END_RUNG wire#w1
   // the same network as SCL:
   #oALARM_FEEDER_NOT_READY_LN_2 := (#DATA.START_LINE_2 AND #iFEEDER_PROFINET_MODE_ACTIVE AND NOT #iPF_INTERLOCK_INPUTS.i_fFeederReady_Line2) OR (#oALARM_FEEDER_NOT_READY_LN_2 AND NOT "DB2120_MPP_ITC_IPC".RESET_FAULTS);
END_REGION

REGION Network 68: CARRIER GAS FLOW BELOW LOW LIMIT FAULT LINE 1 (WARNING)
   RUNG wire#powerrail
      Contact( #iPF_INTERLOCK_INPUTS.i_fWarningFromPF_Line1 )
      Contact( #iPF_INTERLOCK_INPUTS.i_fCarriergasLeL_Line1 )
      Coil( #oWARNING_GAS_FLOW_UNDER_LIMIT_LN_1 )
   END_RUNG
   // the same network as SCL:
   #oWARNING_GAS_FLOW_UNDER_LIMIT_LN_1 := #iPF_INTERLOCK_INPUTS.i_fWarningFromPF_Line1 AND #iPF_INTERLOCK_INPUTS.i_fCarriergasLeL_Line1;
END_REGION

REGION Network 69: CARRIER GAS FLOW BELOW LOW LIMIT FAULT LINE 2 (WARNING)
   RUNG wire#powerrail
      Contact( #iPF_INTERLOCK_INPUTS.i_fWarningFromPF_Line2 )
      Contact( #iPF_INTERLOCK_INPUTS.i_fCarriergasLeL_Line2 )
      Coil( #oWARNING_GAS_FLOW_UNDER_LIMIT_LN_2 )
   END_RUNG
   // the same network as SCL:
   #oWARNING_GAS_FLOW_UNDER_LIMIT_LN_2 := #iPF_INTERLOCK_INPUTS.i_fWarningFromPF_Line2 AND #iPF_INTERLOCK_INPUTS.i_fCarriergasLeL_Line2;
END_REGION

REGION Network 70: DISK SPEED FLOW BELOW LOW LIMIT FAULT LINE 1 (WARNING)
   RUNG wire#powerrail
      Contact( #iPF_INTERLOCK_INPUTS.i_fWarningFromPF_Line1 )
      Contact( #iPF_INTERLOCK_INPUTS.i_fDiskSpeedLeL_Line1 )
      Coil( #oWARNING_DISK_SPEED_UNDER_LIMIT_LN_1 )
   END_RUNG
   // the same network as SCL:
   #oWARNING_DISK_SPEED_UNDER_LIMIT_LN_1 := #iPF_INTERLOCK_INPUTS.i_fWarningFromPF_Line1 AND #iPF_INTERLOCK_INPUTS.i_fDiskSpeedLeL_Line1;
END_REGION

REGION Network 71: DISK SPEED FLOW BELOW LOW LIMIT FAULT LINE 2 (WARNING)
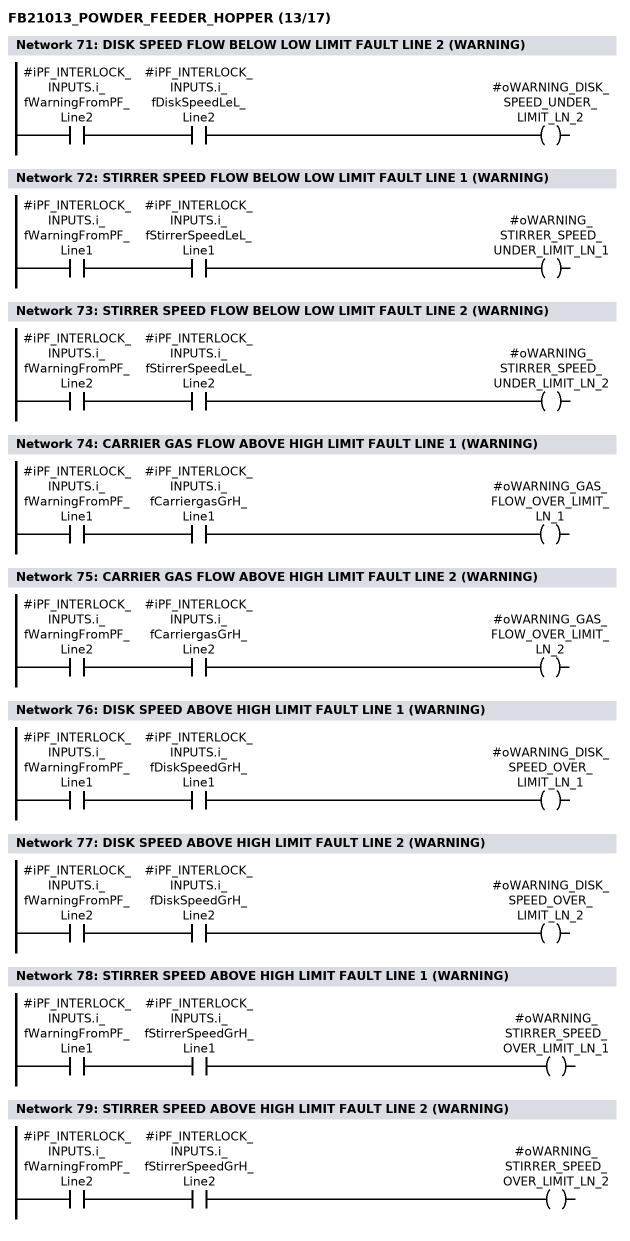
   RUNG wire#powerrail
      Contact( #iPF_INTERLOCK_INPUTS.i_fWarningFromPF_Line2 )
      Contact( #iPF_INTERLOCK_INPUTS.i_fDiskSpeedLeL_Line2 )
      Coil( #oWARNING_DISK_SPEED_UNDER_LIMIT_LN_2 )
   END_RUNG
   // the same network as SCL:
   #oWARNING_DISK_SPEED_UNDER_LIMIT_LN_2 := #iPF_INTERLOCK_INPUTS.i_fWarningFromPF_Line2 AND #iPF_INTERLOCK_INPUTS.i_fDiskSpeedLeL_Line2;
END_REGION

REGION Network 72: STIRRER SPEED FLOW BELOW LOW LIMIT FAULT LINE 1 (WARNING)
   RUNG wire#powerrail
      Contact( #iPF_INTERLOCK_INPUTS.i_fWarningFromPF_Line1 )
      Contact( #iPF_INTERLOCK_INPUTS.i_fStirrerSpeedLeL_Line1 )
      Coil( #oWARNING_STIRRER_SPEED_UNDER_LIMIT_LN_1 )
   END_RUNG
   // the same network as SCL:
   #oWARNING_STIRRER_SPEED_UNDER_LIMIT_LN_1 := #iPF_INTERLOCK_INPUTS.i_fWarningFromPF_Line1 AND #iPF_INTERLOCK_INPUTS.i_fStirrerSpeedLeL_Line1;
END_REGION

REGION Network 73: STIRRER SPEED FLOW BELOW LOW LIMIT FAULT LINE 2 (WARNING)
   RUNG wire#powerrail
      Contact( #iPF_INTERLOCK_INPUTS.i_fWarningFromPF_Line2 )
      Contact( #iPF_INTERLOCK_INPUTS.i_fStirrerSpeedLeL_Line2 )
      Coil( #oWARNING_STIRRER_SPEED_UNDER_LIMIT_LN_2 )
   END_RUNG
   // the same network as SCL:
   #oWARNING_STIRRER_SPEED_UNDER_LIMIT_LN_2 := #iPF_INTERLOCK_INPUTS.i_fWarningFromPF_Line2 AND #iPF_INTERLOCK_INPUTS.i_fStirrerSpeedLeL_Line2;
END_REGION

REGION Network 74: CARRIER GAS FLOW ABOVE HIGH LIMIT FAULT LINE 1 (WARNING)
   RUNG wire#powerrail
      Contact( #iPF_INTERLOCK_INPUTS.i_fWarningFromPF_Line1 )
      Contact( #iPF_INTERLOCK_INPUTS.i_fCarriergasGrH_Line1 )
      Coil( #oWARNING_GAS_FLOW_OVER_LIMIT_LN_1 )
   END_RUNG
   // the same network as SCL:
   #oWARNING_GAS_FLOW_OVER_LIMIT_LN_1 := #iPF_INTERLOCK_INPUTS.i_fWarningFromPF_Line1 AND #iPF_INTERLOCK_INPUTS.i_fCarriergasGrH_Line1;
END_REGION

REGION Network 75: CARRIER GAS FLOW ABOVE HIGH LIMIT FAULT LINE 2 (WARNING)
   RUNG wire#powerrail
      Contact( #iPF_INTERLOCK_INPUTS.i_fWarningFromPF_Line2 )
      Contact( #iPF_INTERLOCK_INPUTS.i_fCarriergasGrH_Line2 )
      Coil( #oWARNING_GAS_FLOW_OVER_LIMIT_LN_2 )
   END_RUNG
   // the same network as SCL:
   #oWARNING_GAS_FLOW_OVER_LIMIT_LN_2 := #iPF_INTERLOCK_INPUTS.i_fWarningFromPF_Line2 AND #iPF_INTERLOCK_INPUTS.i_fCarriergasGrH_Line2;
END_REGION

REGION Network 76: DISK SPEED ABOVE HIGH LIMIT FAULT LINE 1 (WARNING)
   RUNG wire#powerrail
      Contact( #iPF_INTERLOCK_INPUTS.i_fWarningFromPF_Line1 )
      Contact( #iPF_INTERLOCK_INPUTS.i_fDiskSpeedGrH_Line1 )
      Coil( #oWARNING_DISK_SPEED_OVER_LIMIT_LN_1 )
   END_RUNG
   // the same network as SCL:
   #oWARNING_DISK_SPEED_OVER_LIMIT_LN_1 := #iPF_INTERLOCK_INPUTS.i_fWarningFromPF_Line1 AND #iPF_INTERLOCK_INPUTS.i_fDiskSpeedGrH_Line1;
END_REGION

REGION Network 77: DISK SPEED ABOVE HIGH LIMIT FAULT LINE 2 (WARNING)
   RUNG wire#powerrail
      Contact( #iPF_INTERLOCK_INPUTS.i_fWarningFromPF_Line2 )
      Contact( #iPF_INTERLOCK_INPUTS.i_fDiskSpeedGrH_Line2 )
      Coil( #oWARNING_DISK_SPEED_OVER_LIMIT_LN_2 )
   END_RUNG
   // the same network as SCL:
   #oWARNING_DISK_SPEED_OVER_LIMIT_LN_2 := #iPF_INTERLOCK_INPUTS.i_fWarningFromPF_Line2 AND #iPF_INTERLOCK_INPUTS.i_fDiskSpeedGrH_Line2;
END_REGION

REGION Network 78: STIRRER SPEED ABOVE HIGH LIMIT FAULT LINE 1 (WARNING)
   RUNG wire#powerrail
      Contact( #iPF_INTERLOCK_INPUTS.i_fWarningFromPF_Line1 )
      Contact( #iPF_INTERLOCK_INPUTS.i_fStirrerSpeedGrH_Line1 )
      Coil( #oWARNING_STIRRER_SPEED_OVER_LIMIT_LN_1 )
   END_RUNG
   // the same network as SCL:
   #oWARNING_STIRRER_SPEED_OVER_LIMIT_LN_1 := #iPF_INTERLOCK_INPUTS.i_fWarningFromPF_Line1 AND #iPF_INTERLOCK_INPUTS.i_fStirrerSpeedGrH_Line1;
END_REGION

REGION Network 79: STIRRER SPEED ABOVE HIGH LIMIT FAULT LINE 2 (WARNING)
   RUNG wire#powerrail
      Contact( #iPF_INTERLOCK_INPUTS.i_fWarningFromPF_Line2 )
      Contact( #iPF_INTERLOCK_INPUTS.i_fStirrerSpeedGrH_Line2 )
      Coil( #oWARNING_STIRRER_SPEED_OVER_LIMIT_LN_2 )
   END_RUNG
   // the same network as SCL:
   #oWARNING_STIRRER_SPEED_OVER_LIMIT_LN_2 := #iPF_INTERLOCK_INPUTS.i_fWarningFromPF_Line2 AND #iPF_INTERLOCK_INPUTS.i_fStirrerSpeedGrH_Line2;
END_REGION

REGION Network 80: IMMEDIATE STOP ALARMS
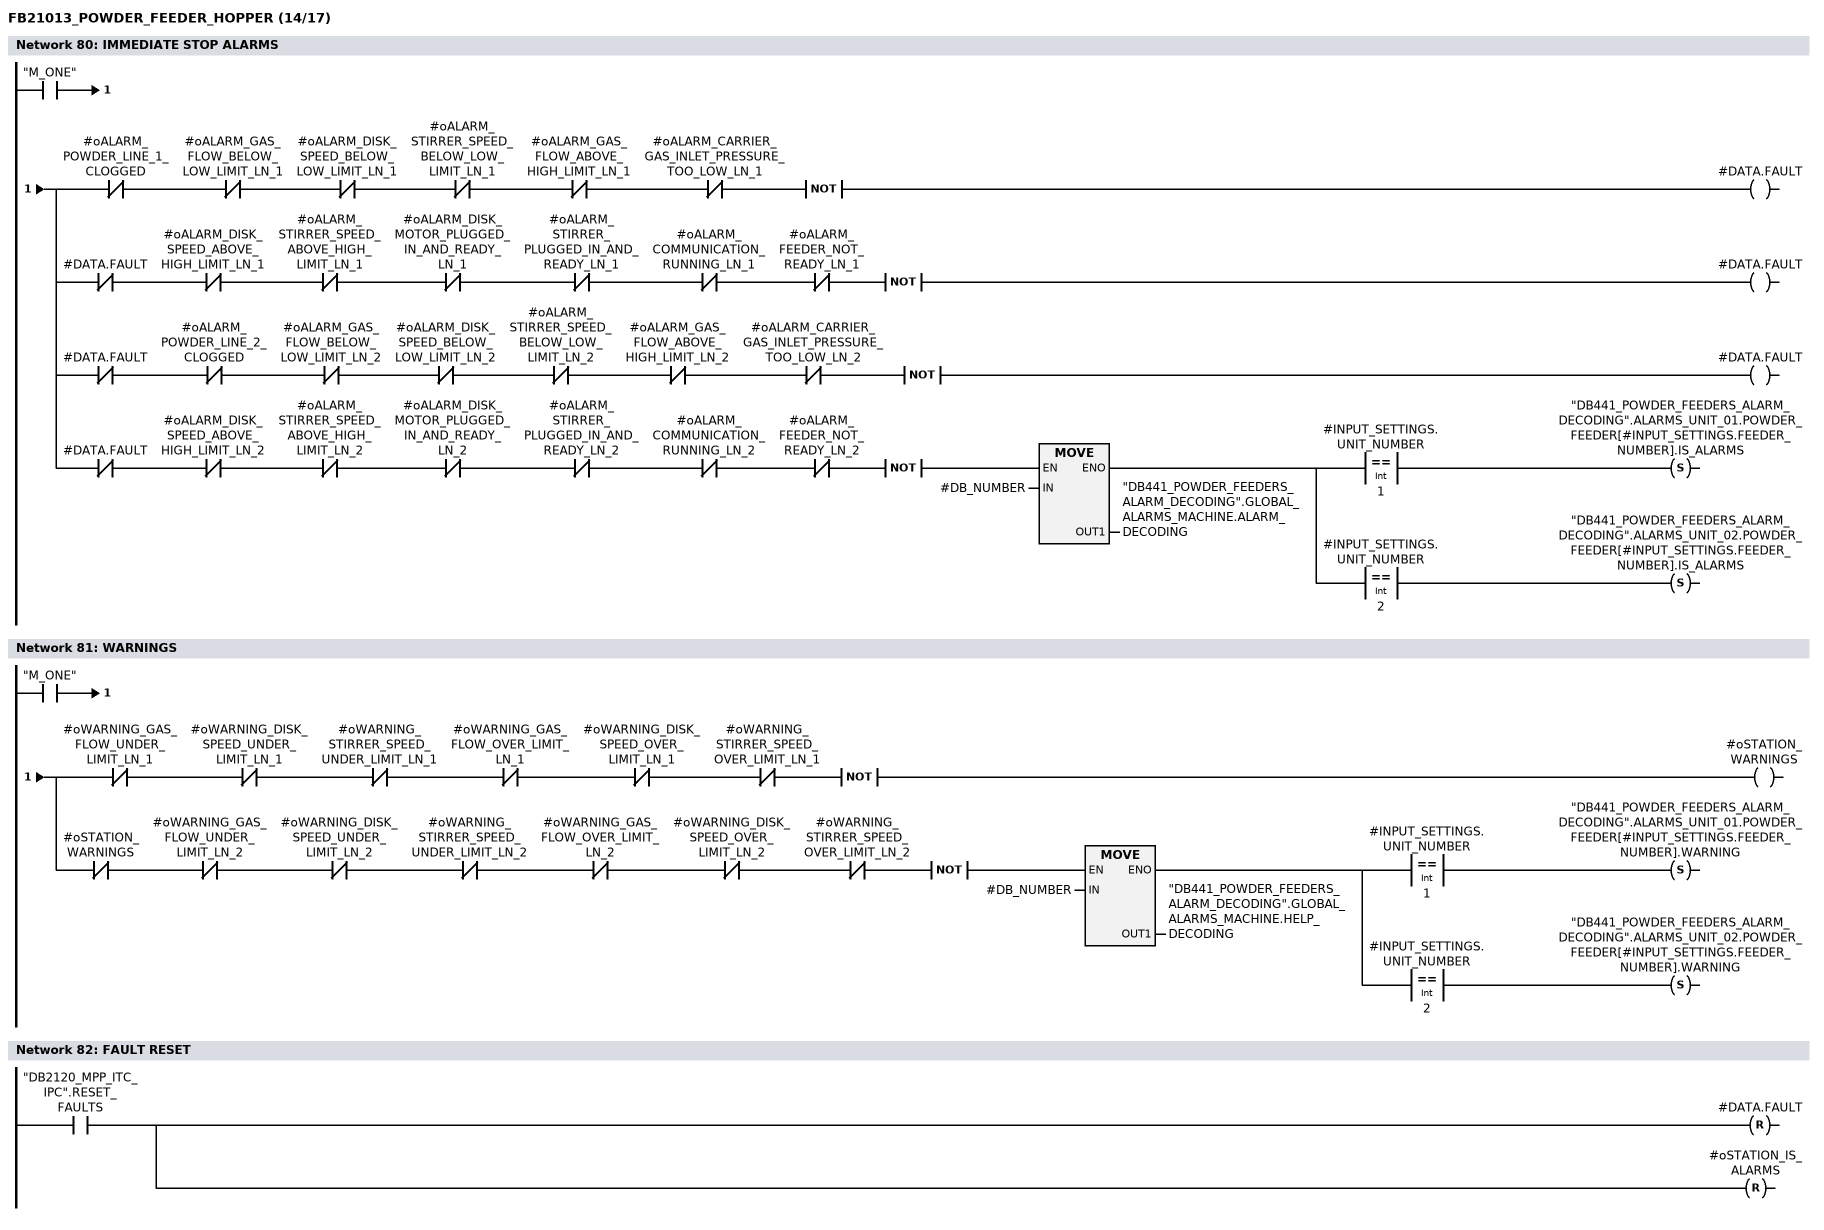
   RUNG wire#powerrail
      Contact( "M_ONE" )
      wire#w1
      I_Contact( #oALARM_POWDER_LINE_1_CLOGGED )
      I_Contact( #oALARM_GAS_FLOW_BELOW_LOW_LIMIT_LN_1 )
      I_Contact( #oALARM_DISK_SPEED_BELOW_LOW_LIMIT_LN_1 )
      I_Contact( #oALARM_STIRRER_SPEED_BELOW_LOW_LIMIT_LN_1 )
      I_Contact( #oALARM_GAS_FLOW_ABOVE_HIGH_LIMIT_LN_1 )
      I_Contact( #oALARM_CARRIER_GAS_INLET_PRESSURE_TOO_LOW_LN_1 )
      Not()
      Coil( #DATA.FAULT )
   END_RUNG
   RUNG wire#w1
      I_Contact( #DATA.FAULT )
      I_Contact( #oALARM_DISK_SPEED_ABOVE_HIGH_LIMIT_LN_1 )
      I_Contact( #oALARM_STIRRER_SPEED_ABOVE_HIGH_LIMIT_LN_1 )
      I_Contact( #oALARM_DISK_MOTOR_PLUGGED_IN_AND_READY_LN_1 )
      I_Contact( #oALARM_STIRRER_PLUGGED_IN_AND_READY_LN_1 )
      I_Contact( #oALARM_COMMUNICATION_RUNNING_LN_1 )
      I_Contact( #oALARM_FEEDER_NOT_READY_LN_1 )
      Not()
      Coil( #DATA.FAULT )
   END_RUNG
   RUNG wire#w1
      I_Contact( #DATA.FAULT )
      I_Contact( #oALARM_POWDER_LINE_2_CLOGGED )
      I_Contact( #oALARM_GAS_FLOW_BELOW_LOW_LIMIT_LN_2 )
      I_Contact( #oALARM_DISK_SPEED_BELOW_LOW_LIMIT_LN_2 )
      I_Contact( #oALARM_STIRRER_SPEED_BELOW_LOW_LIMIT_LN_2 )
      I_Contact( #oALARM_GAS_FLOW_ABOVE_HIGH_LIMIT_LN_2 )
      I_Contact( #oALARM_CARRIER_GAS_INLET_PRESSURE_TOO_LOW_LN_2 )
      Not()
      Coil( #DATA.FAULT )
   END_RUNG
   RUNG wire#w1
      I_Contact( #DATA.FAULT )
      I_Contact( #oALARM_DISK_SPEED_ABOVE_HIGH_LIMIT_LN_2 )
      I_Contact( #oALARM_STIRRER_SPEED_ABOVE_HIGH_LIMIT_LN_2 )
      I_Contact( #oALARM_DISK_MOTOR_PLUGGED_IN_AND_READY_LN_2 )
      I_Contact( #oALARM_STIRRER_PLUGGED_IN_AND_READY_LN_2 )
      I_Contact( #oALARM_COMMUNICATION_RUNNING_LN_2 )
      I_Contact( #oALARM_FEEDER_NOT_READY_LN_2 )
      Not()
      Move(in := #DB_NUMBER, out1 => "DB441_POWDER_FEEDERS_ALARM_DECODING".GLOBAL_ALARMS_MACHINE.ALARM_DECODING)
      wire#w2
      { S7_Templates := "SrcType := Int" } EQ_Contact(in1 := #INPUT_SETTINGS.UNIT_NUMBER, in2 := 1)
      S_Coil( "DB441_POWDER_FEEDERS_ALARM_DECODING".ALARMS_UNIT_01.POWDER_FEEDER[#INPUT_SETTINGS.FEEDER_NUMBER].IS_ALARMS )
   END_RUNG
   RUNG wire#w2
      { S7_Templates := "SrcType := Int" } EQ_Contact(in1 := #INPUT_SETTINGS.UNIT_NUMBER, in2 := 2)
      S_Coil( "DB441_POWDER_FEEDERS_ALARM_DECODING".ALARMS_UNIT_02.POWDER_FEEDER[#INPUT_SETTINGS.FEEDER_NUMBER].IS_ALARMS )
   END_RUNG
   // the same network as SCL:
   #DATA.FAULT := NOT ("M_ONE" AND NOT #oALARM_POWDER_LINE_1_CLOGGED AND NOT #oALARM_GAS_FLOW_BELOW_LOW_LIMIT_LN_1 AND NOT #oALARM_DISK_SPEED_BELOW_LOW_LIMIT_LN_1 AND NOT #oALARM_STIRRER_SPEED_BELOW_LOW_LIMIT_LN_1 AND NOT #oALARM_GAS_FLOW_ABOVE_HIGH_LIMIT_LN_1 AND NOT #oALARM_CARRIER_GAS_INLET_PRESSURE_TOO_LOW_LN_1);
   #DATA.FAULT := NOT ("M_ONE" AND NOT #DATA.FAULT AND NOT #oALARM_DISK_SPEED_ABOVE_HIGH_LIMIT_LN_1 AND NOT #oALARM_STIRRER_SPEED_ABOVE_HIGH_LIMIT_LN_1 AND NOT #oALARM_DISK_MOTOR_PLUGGED_IN_AND_READY_LN_1 AND NOT #oALARM_STIRRER_PLUGGED_IN_AND_READY_LN_1 AND NOT #oALARM_COMMUNICATION_RUNNING_LN_1 AND NOT #oALARM_FEEDER_NOT_READY_LN_1);
   #DATA.FAULT := NOT ("M_ONE" AND NOT #DATA.FAULT AND NOT #oALARM_POWDER_LINE_2_CLOGGED AND NOT #oALARM_GAS_FLOW_BELOW_LOW_LIMIT_LN_2 AND NOT #oALARM_DISK_SPEED_BELOW_LOW_LIMIT_LN_2 AND NOT #oALARM_STIRRER_SPEED_BELOW_LOW_LIMIT_LN_2 AND NOT #oALARM_GAS_FLOW_ABOVE_HIGH_LIMIT_LN_2 AND NOT #oALARM_CARRIER_GAS_INLET_PRESSURE_TOO_LOW_LN_2);
   #_w1 := NOT ("M_ONE" AND NOT #DATA.FAULT AND NOT #oALARM_DISK_SPEED_ABOVE_HIGH_LIMIT_LN_2 AND NOT #oALARM_STIRRER_SPEED_ABOVE_HIGH_LIMIT_LN_2 AND NOT #oALARM_DISK_MOTOR_PLUGGED_IN_AND_READY_LN_2 AND NOT #oALARM_STIRRER_PLUGGED_IN_AND_READY_LN_2 AND NOT #oALARM_COMMUNICATION_RUNNING_LN_2 AND NOT #oALARM_FEEDER_NOT_READY_LN_2);
   IF #_w1 THEN
       "DB441_POWDER_FEEDERS_ALARM_DECODING".GLOBAL_ALARMS_MACHINE.ALARM_DECODING := #DB_NUMBER;
   END_IF;
   IF #_w1 AND (#INPUT_SETTINGS.UNIT_NUMBER = 1) THEN
       "DB441_POWDER_FEEDERS_ALARM_DECODING".ALARMS_UNIT_01.POWDER_FEEDER[#INPUT_SETTINGS.FEEDER_NUMBER].IS_ALARMS := TRUE;
   END_IF;
   IF #_w1 AND (#INPUT_SETTINGS.UNIT_NUMBER = 2) THEN
       "DB441_POWDER_FEEDERS_ALARM_DECODING".ALARMS_UNIT_02.POWDER_FEEDER[#INPUT_SETTINGS.FEEDER_NUMBER].IS_ALARMS := TRUE;
   END_IF;
END_REGION

REGION Network 81: WARNINGS
   RUNG wire#powerrail
      Contact( "M_ONE" )
      wire#w1
      I_Contact( #oWARNING_GAS_FLOW_UNDER_LIMIT_LN_1 )
      I_Contact( #oWARNING_DISK_SPEED_UNDER_LIMIT_LN_1 )
      I_Contact( #oWARNING_STIRRER_SPEED_UNDER_LIMIT_LN_1 )
      I_Contact( #oWARNING_GAS_FLOW_OVER_LIMIT_LN_1 )
      I_Contact( #oWARNING_DISK_SPEED_OVER_LIMIT_LN_1 )
      I_Contact( #oWARNING_STIRRER_SPEED_OVER_LIMIT_LN_1 )
      Not()
      Coil( #oSTATION_WARNINGS )
   END_RUNG
   RUNG wire#w1
      I_Contact( #oSTATION_WARNINGS )
      I_Contact( #oWARNING_GAS_FLOW_UNDER_LIMIT_LN_2 )
      I_Contact( #oWARNING_DISK_SPEED_UNDER_LIMIT_LN_2 )
      I_Contact( #oWARNING_STIRRER_SPEED_UNDER_LIMIT_LN_2 )
      I_Contact( #oWARNING_GAS_FLOW_OVER_LIMIT_LN_2 )
      I_Contact( #oWARNING_DISK_SPEED_OVER_LIMIT_LN_2 )
      I_Contact( #oWARNING_STIRRER_SPEED_OVER_LIMIT_LN_2 )
      Not()
      Move(in := #DB_NUMBER, out1 => "DB441_POWDER_FEEDERS_ALARM_DECODING".GLOBAL_ALARMS_MACHINE.HELP_DECODING)
      wire#w2
      { S7_Templates := "SrcType := Int" } EQ_Contact(in1 := #INPUT_SETTINGS.UNIT_NUMBER, in2 := 1)
      S_Coil( "DB441_POWDER_FEEDERS_ALARM_DECODING".ALARMS_UNIT_01.POWDER_FEEDER[#INPUT_SETTINGS.FEEDER_NUMBER].WARNING )
   END_RUNG
   RUNG wire#w2
      { S7_Templates := "SrcType := Int" } EQ_Contact(in1 := #INPUT_SETTINGS.UNIT_NUMBER, in2 := 2)
      S_Coil( "DB441_POWDER_FEEDERS_ALARM_DECODING".ALARMS_UNIT_02.POWDER_FEEDER[#INPUT_SETTINGS.FEEDER_NUMBER].WARNING )
   END_RUNG
   // the same network as SCL:
   #oSTATION_WARNINGS := NOT ("M_ONE" AND NOT #oWARNING_GAS_FLOW_UNDER_LIMIT_LN_1 AND NOT #oWARNING_DISK_SPEED_UNDER_LIMIT_LN_1 AND NOT #oWARNING_STIRRER_SPEED_UNDER_LIMIT_LN_1 AND NOT #oWARNING_GAS_FLOW_OVER_LIMIT_LN_1 AND NOT #oWARNING_DISK_SPEED_OVER_LIMIT_LN_1 AND NOT #oWARNING_STIRRER_SPEED_OVER_LIMIT_LN_1);
   #_w1 := NOT ("M_ONE" AND NOT #oSTATION_WARNINGS AND NOT #oWARNING_GAS_FLOW_UNDER_LIMIT_LN_2 AND NOT #oWARNING_DISK_SPEED_UNDER_LIMIT_LN_2 AND NOT #oWARNING_STIRRER_SPEED_UNDER_LIMIT_LN_2 AND NOT #oWARNING_GAS_FLOW_OVER_LIMIT_LN_2 AND NOT #oWARNING_DISK_SPEED_OVER_LIMIT_LN_2 AND NOT #oWARNING_STIRRER_SPEED_OVER_LIMIT_LN_2);
   IF #_w1 THEN
       "DB441_POWDER_FEEDERS_ALARM_DECODING".GLOBAL_ALARMS_MACHINE.HELP_DECODING := #DB_NUMBER;
   END_IF;
   IF #_w1 AND (#INPUT_SETTINGS.UNIT_NUMBER = 1) THEN
       "DB441_POWDER_FEEDERS_ALARM_DECODING".ALARMS_UNIT_01.POWDER_FEEDER[#INPUT_SETTINGS.FEEDER_NUMBER].WARNING := TRUE;
   END_IF;
   IF #_w1 AND (#INPUT_SETTINGS.UNIT_NUMBER = 2) THEN
       "DB441_POWDER_FEEDERS_ALARM_DECODING".ALARMS_UNIT_02.POWDER_FEEDER[#INPUT_SETTINGS.FEEDER_NUMBER].WARNING := TRUE;
   END_IF;
END_REGION

REGION Network 82: FAULT RESET
   RUNG wire#powerrail
      Contact( "DB2120_MPP_ITC_IPC".RESET_FAULTS )
      wire#w1
      R_Coil( #DATA.FAULT )
   END_RUNG
   RUNG wire#w1
      R_Coil( #oSTATION_IS_ALARMS )
   END_RUNG
   // the same network as SCL:
   IF "DB2120_MPP_ITC_IPC".RESET_FAULTS THEN
       #DATA.FAULT := FALSE;
       #oSTATION_IS_ALARMS := FALSE;
   END_IF;
END_REGION

REGION Network 83: START GENERAL CONDITIONS HELP
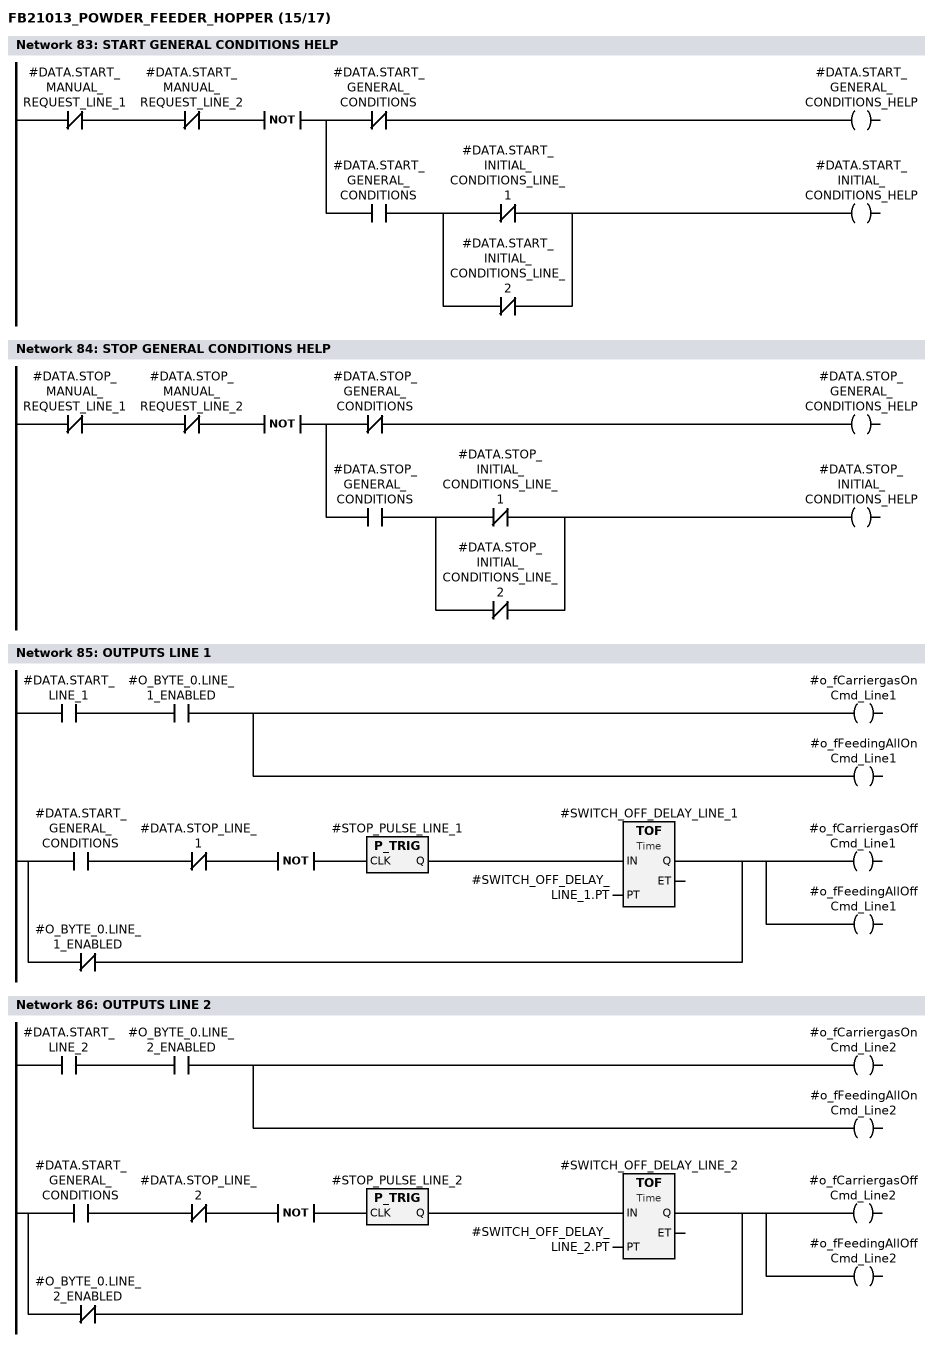
   RUNG wire#powerrail
      I_Contact( #DATA.START_MANUAL_REQUEST_LINE_1 )
      I_Contact( #DATA.START_MANUAL_REQUEST_LINE_2 )
      Not()
      wire#w1
      I_Contact( #DATA.START_GENERAL_CONDITIONS )
      Coil( #DATA.START_GENERAL_CONDITIONS_HELP )
   END_RUNG
   RUNG wire#w1
      Contact( #DATA.START_GENERAL_CONDITIONS )
      wire#w2
      I_Contact( #DATA.START_INITIAL_CONDITIONS_LINE_1 )
      wire#w3
      Coil( #DATA.START_INITIAL_CONDITIONS_HELP )
   END_RUNG
   RUNG wire#w2
      I_Contact( #DATA.START_INITIAL_CONDITIONS_LINE_2 )
   END_RUNG wire#w3
   // the same network as SCL:
   #_w1 := NOT (NOT #DATA.START_MANUAL_REQUEST_LINE_1 AND NOT #DATA.START_MANUAL_REQUEST_LINE_2);
   #DATA.START_GENERAL_CONDITIONS_HELP := #_w1 AND NOT #DATA.START_GENERAL_CONDITIONS;
   #DATA.START_INITIAL_CONDITIONS_HELP := #_w1 AND #DATA.START_GENERAL_CONDITIONS AND (NOT #DATA.START_INITIAL_CONDITIONS_LINE_1 OR NOT #DATA.START_INITIAL_CONDITIONS_LINE_2);
END_REGION

REGION Network 84: STOP GENERAL CONDITIONS HELP
   RUNG wire#powerrail
      I_Contact( #DATA.STOP_MANUAL_REQUEST_LINE_1 )
      I_Contact( #DATA.STOP_MANUAL_REQUEST_LINE_2 )
      Not()
      wire#w1
      I_Contact( #DATA.STOP_GENERAL_CONDITIONS )
      Coil( #DATA.STOP_GENERAL_CONDITIONS_HELP )
   END_RUNG
   RUNG wire#w1
      Contact( #DATA.STOP_GENERAL_CONDITIONS )
      wire#w2
      I_Contact( #DATA.STOP_INITIAL_CONDITIONS_LINE_1 )
      wire#w3
      Coil( #DATA.STOP_INITIAL_CONDITIONS_HELP )
   END_RUNG
   RUNG wire#w2
      I_Contact( #DATA.STOP_INITIAL_CONDITIONS_LINE_2 )
   END_RUNG wire#w3
   // the same network as SCL:
   #_w1 := NOT (NOT #DATA.STOP_MANUAL_REQUEST_LINE_1 AND NOT #DATA.STOP_MANUAL_REQUEST_LINE_2);
   #DATA.STOP_GENERAL_CONDITIONS_HELP := #_w1 AND NOT #DATA.STOP_GENERAL_CONDITIONS;
   #DATA.STOP_INITIAL_CONDITIONS_HELP := #_w1 AND #DATA.STOP_GENERAL_CONDITIONS AND (NOT #DATA.STOP_INITIAL_CONDITIONS_LINE_1 OR NOT #DATA.STOP_INITIAL_CONDITIONS_LINE_2);
END_REGION

REGION Network 85: OUTPUTS LINE 1
   RUNG wire#powerrail
      Contact( #DATA.START_LINE_1 )
      Contact( #O_BYTE_0.LINE_1_ENABLED )
      wire#w1
      Coil( #o_fCarriergasOnCmd_Line1 )
   END_RUNG
   RUNG wire#w1
      Coil( #o_fFeedingAllOnCmd_Line1 )
   END_RUNG
   RUNG wire#powerrail
      Contact( #DATA.START_GENERAL_CONDITIONS )
      I_Contact( #DATA.STOP_LINE_1 )
      Not()
      P_Trig( #STOP_PULSE_LINE_1 )
      { S7_Templates := "time_type := Time" } #SWITCH_OFF_DELAY_LINE_1.TOF(pt := #SWITCH_OFF_DELAY_LINE_1.PT, et =>)
      wire#w2
      Coil( #o_fCarriergasOffCmd_Line1 )
   END_RUNG
   RUNG wire#powerrail
      I_Contact( #O_BYTE_0.LINE_1_ENABLED )
   END_RUNG wire#w2
   RUNG wire#w2
      Coil( #o_fFeedingAllOffCmd_Line1 )
   END_RUNG
   // the same network as SCL:
   #o_fCarriergasOnCmd_Line1 := #DATA.START_LINE_1 AND #O_BYTE_0.LINE_1_ENABLED;
   #o_fFeedingAllOnCmd_Line1 := #o_fCarriergasOnCmd_Line1;
   #_w1 := NOT (#DATA.START_GENERAL_CONDITIONS AND NOT #DATA.STOP_LINE_1);
   #_w2 := #_w1 AND NOT #STOP_PULSE_LINE_1;   // rising edge
   #STOP_PULSE_LINE_1 := #_w1;
   #SWITCH_OFF_DELAY_LINE_1(IN := #_w2, PT := #SWITCH_OFF_DELAY_LINE_1.PT);   // TOF
   #o_fCarriergasOffCmd_Line1 := #SWITCH_OFF_DELAY_LINE_1.Q OR NOT #O_BYTE_0.LINE_1_ENABLED;
   #o_fFeedingAllOffCmd_Line1 := #o_fCarriergasOffCmd_Line1;
END_REGION

REGION Network 86: OUTPUTS LINE 2
   RUNG wire#powerrail
      Contact( #DATA.START_LINE_2 )
      Contact( #O_BYTE_0.LINE_2_ENABLED )
      wire#w1
      Coil( #o_fCarriergasOnCmd_Line2 )
   END_RUNG
   RUNG wire#w1
      Coil( #o_fFeedingAllOnCmd_Line2 )
   END_RUNG
   RUNG wire#powerrail
      Contact( #DATA.START_GENERAL_CONDITIONS )
      I_Contact( #DATA.STOP_LINE_2 )
      Not()
      P_Trig( #STOP_PULSE_LINE_2 )
      { S7_Templates := "time_type := Time" } #SWITCH_OFF_DELAY_LINE_2.TOF(pt := #SWITCH_OFF_DELAY_LINE_2.PT, et =>)
      wire#w2
      Coil( #o_fCarriergasOffCmd_Line2 )
   END_RUNG
   RUNG wire#powerrail
      I_Contact( #O_BYTE_0.LINE_2_ENABLED )
   END_RUNG wire#w2
   RUNG wire#w2
      Coil( #o_fFeedingAllOffCmd_Line2 )
   END_RUNG
   // the same network as SCL:
   #o_fCarriergasOnCmd_Line2 := #DATA.START_LINE_2 AND #O_BYTE_0.LINE_2_ENABLED;
   #o_fFeedingAllOnCmd_Line2 := #o_fCarriergasOnCmd_Line2;
   #_w1 := NOT (#DATA.START_GENERAL_CONDITIONS AND NOT #DATA.STOP_LINE_2);
   #_w2 := #_w1 AND NOT #STOP_PULSE_LINE_2;   // rising edge
   #STOP_PULSE_LINE_2 := #_w1;
   #SWITCH_OFF_DELAY_LINE_2(IN := #_w2, PT := #SWITCH_OFF_DELAY_LINE_2.PT);   // TOF
   #o_fCarriergasOffCmd_Line2 := #SWITCH_OFF_DELAY_LINE_2.Q OR NOT #O_BYTE_0.LINE_2_ENABLED;
   #o_fFeedingAllOffCmd_Line2 := #o_fCarriergasOffCmd_Line2;
END_REGION

REGION Network 87: SHUTDOWN
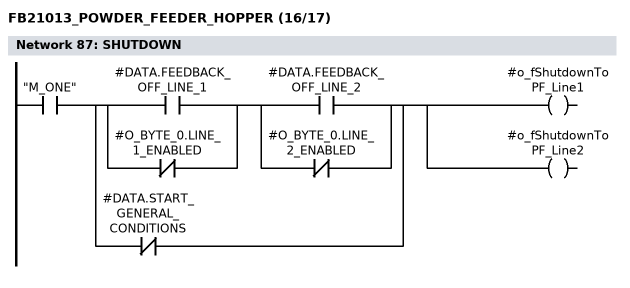
   RUNG wire#powerrail
      Contact( "M_ONE" )
      wire#w1
      Contact( #DATA.FEEDBACK_OFF_LINE_1 )
      wire#w2
      Contact( #DATA.FEEDBACK_OFF_LINE_2 )
      wire#w3
      Coil( #o_fShutdownToPF_Line1 )
   END_RUNG
   RUNG wire#w1
      I_Contact( #O_BYTE_0.LINE_1_ENABLED )
   END_RUNG wire#w2
   RUNG wire#w2
      I_Contact( #O_BYTE_0.LINE_2_ENABLED )
   END_RUNG wire#w3
   RUNG wire#w1
      I_Contact( #DATA.START_GENERAL_CONDITIONS )
   END_RUNG wire#w3
   RUNG wire#w3
      Coil( #o_fShutdownToPF_Line2 )
   END_RUNG
   // the same network as SCL:
   #o_fShutdownToPF_Line1 := "M_ONE" AND (((#DATA.FEEDBACK_OFF_LINE_1 OR NOT #O_BYTE_0.LINE_1_ENABLED) AND (#DATA.FEEDBACK_OFF_LINE_2 OR NOT #O_BYTE_0.LINE_2_ENABLED)) OR NOT #DATA.START_GENERAL_CONDITIONS);
   #o_fShutdownToPF_Line2 := #o_fShutdownToPF_Line1;
END_REGION

REGION Network 88: HOPPER STATUS
   // STATUS:
   // 0: OFF WITH NO CONDITIONS
   // 1: ON
   // 2: OFF WITH CONDITIONS TO SWITCH ON
   // 3: SWITCH ON SEQUENCE RUNNING
   // 4: SWITCH OFF SEQUENCE RUNNING
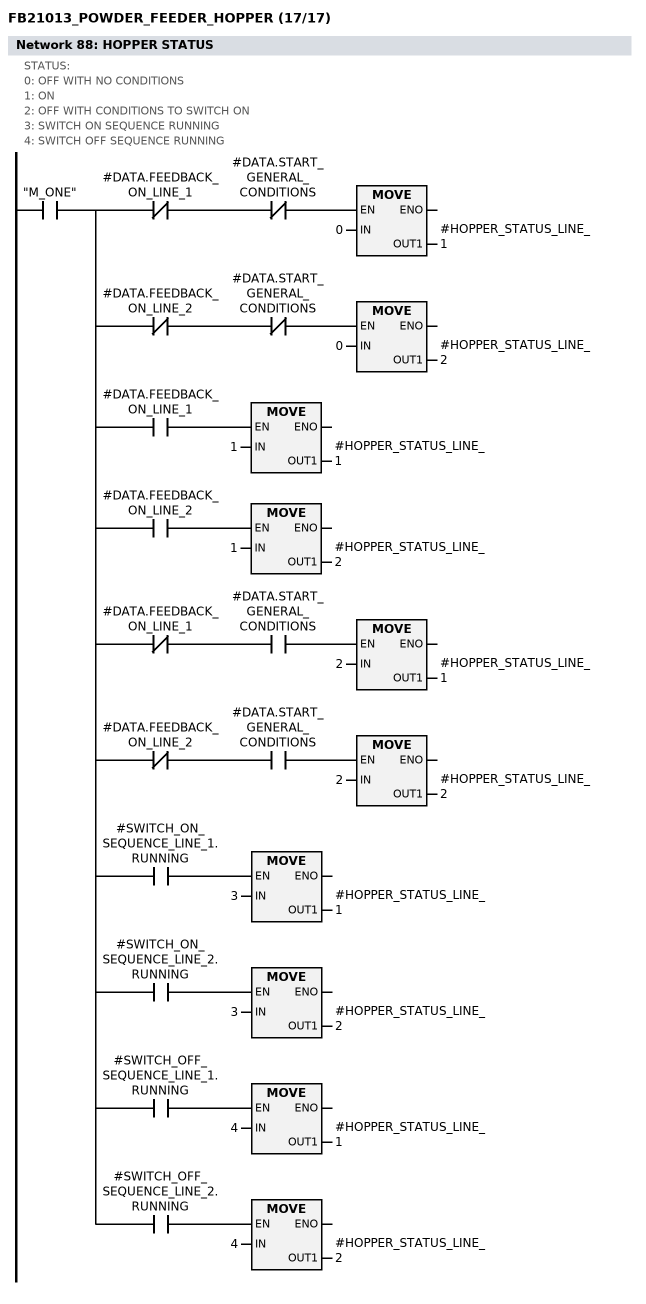
   RUNG wire#powerrail
      Contact( "M_ONE" )
      wire#w1
      I_Contact( #DATA.FEEDBACK_ON_LINE_1 )
      I_Contact( #DATA.START_GENERAL_CONDITIONS )
      Move(in := 0, out1 => #HOPPER_STATUS_LINE_1)
   END_RUNG
   RUNG wire#w1
      I_Contact( #DATA.FEEDBACK_ON_LINE_2 )
      I_Contact( #DATA.START_GENERAL_CONDITIONS )
      Move(in := 0, out1 => #HOPPER_STATUS_LINE_2)
   END_RUNG
   RUNG wire#w1
      Contact( #DATA.FEEDBACK_ON_LINE_1 )
      Move(in := 1, out1 => #HOPPER_STATUS_LINE_1)
   END_RUNG
   RUNG wire#w1
      Contact( #DATA.FEEDBACK_ON_LINE_2 )
      Move(in := 1, out1 => #HOPPER_STATUS_LINE_2)
   END_RUNG
   RUNG wire#w1
      I_Contact( #DATA.FEEDBACK_ON_LINE_1 )
      Contact( #DATA.START_GENERAL_CONDITIONS )
      Move(in := 2, out1 => #HOPPER_STATUS_LINE_1)
   END_RUNG
   RUNG wire#w1
      I_Contact( #DATA.FEEDBACK_ON_LINE_2 )
      Contact( #DATA.START_GENERAL_CONDITIONS )
      Move(in := 2, out1 => #HOPPER_STATUS_LINE_2)
   END_RUNG
   RUNG wire#w1
      Contact( #SWITCH_ON_SEQUENCE_LINE_1.RUNNING )
      Move(in := 3, out1 => #HOPPER_STATUS_LINE_1)
   END_RUNG
   RUNG wire#w1
      Contact( #SWITCH_ON_SEQUENCE_LINE_2.RUNNING )
      Move(in := 3, out1 => #HOPPER_STATUS_LINE_2)
   END_RUNG
   RUNG wire#w1
      Contact( #SWITCH_OFF_SEQUENCE_LINE_1.RUNNING )
      Move(in := 4, out1 => #HOPPER_STATUS_LINE_1)
   END_RUNG
   RUNG wire#w1
      Contact( #SWITCH_OFF_SEQUENCE_LINE_2.RUNNING )
      Move(in := 4, out1 => #HOPPER_STATUS_LINE_2)
   END_RUNG
   // the same network as SCL:
   IF "M_ONE" AND NOT #DATA.FEEDBACK_ON_LINE_1 AND NOT #DATA.START_GENERAL_CONDITIONS THEN
       #HOPPER_STATUS_LINE_1 := 0;
   END_IF;
   IF "M_ONE" AND NOT #DATA.FEEDBACK_ON_LINE_2 AND NOT #DATA.START_GENERAL_CONDITIONS THEN
       #HOPPER_STATUS_LINE_2 := 0;
   END_IF;
   IF "M_ONE" AND #DATA.FEEDBACK_ON_LINE_1 THEN #HOPPER_STATUS_LINE_1 := 1; END_IF;
   IF "M_ONE" AND #DATA.FEEDBACK_ON_LINE_2 THEN #HOPPER_STATUS_LINE_2 := 1; END_IF;
   IF "M_ONE" AND NOT #DATA.FEEDBACK_ON_LINE_1 AND #DATA.START_GENERAL_CONDITIONS THEN
       #HOPPER_STATUS_LINE_1 := 2;
   END_IF;
   IF "M_ONE" AND NOT #DATA.FEEDBACK_ON_LINE_2 AND #DATA.START_GENERAL_CONDITIONS THEN
       #HOPPER_STATUS_LINE_2 := 2;
   END_IF;
   IF "M_ONE" AND #SWITCH_ON_SEQUENCE_LINE_1.RUNNING THEN #HOPPER_STATUS_LINE_1 := 3; END_IF;
   IF "M_ONE" AND #SWITCH_ON_SEQUENCE_LINE_2.RUNNING THEN #HOPPER_STATUS_LINE_2 := 3; END_IF;
   IF "M_ONE" AND #SWITCH_OFF_SEQUENCE_LINE_1.RUNNING THEN #HOPPER_STATUS_LINE_1 := 4; END_IF;
   IF "M_ONE" AND #SWITCH_OFF_SEQUENCE_LINE_2.RUNNING THEN #HOPPER_STATUS_LINE_2 := 4; END_IF;
END_REGION
END_FUNCTION_BLOCK
